C07218=1044.271,328.276,-116.998,172.493,41.338,157.946
C07219=1044.264,328.029,-116.963,172.488,41.335,157.945
C07220=1044.256,327.782,-116.928,172.484,41.332,157.944
C07221=1044.249,327.534,-116.893,172.479,41.328,157.943
C07222=1044.242,327.286,-116.857,172.474,41.325,157.942
C07223=1044.235,327.039,-116.823,172.470,41.322,157.941
C07224=1044.227,326.791,-116.787,172.466,41.319,157.940
C07225=1044.220,326.544,-116.753,172.461,41.316,157.939
C07226=1044.213,326.297,-116.718,172.457,41.313,157.938
C07227=1044.206,326.049,-116.683,172.453,41.310,157.937
C07228=1044.198,325.802,-116.648,172.449,41.307,157.936
C07229=1044.191,325.554,-116.613,172.444,41.304,157.935
C07230=1044.184,325.307,-116.578,172.440,41.301,157.934
C07231=1044.177,325.060,-116.543,172.436,41.298,157.933
C07232=1044.170,324.812,-116.509,172.431,41.295,157.932
C07233=1044.163,324.564,-116.474,172.427,41.292,157.931
C07234=1044.156,324.317,-116.438,172.423,41.289,157.930
C07235=1044.148,324.070,-116.404,172.419,41.286,157.929
C07236=1044.141,323.822,-116.369,172.414,41.283,157.929
C07237=1044.134,323.575,-116.335,172.410,41.280,157.928
C07238=1044.128,323.327,-116.300,172.406,41.277,157.927
C07239=1044.120,323.080,-116.265,172.401,41.274,157.926
C07240=1044.113,322.833,-116.230,172.398,41.271,157.925
C07241=1044.106,322.584,-116.195,172.392,41.268,157.924
C07242=1044.099,322.337,-116.161,172.388,41.265,157.923
C07243=1044.092,322.090,-116.126,172.384,41.262,157.922
C07244=1044.085,321.842,-116.092,172.380,41.259,157.921
C07245=1044.078,321.595,-116.057,172.376,41.256,157.920
C07246=1044.071,321.347,-116.023,172.371,41.254,157.920
C07247=1044.064,321.100,-115.988,172.367,41.250,157.919
C07248=1044.056,320.853,-115.953,172.363,41.247,157.918
C07249=1044.050,320.605,-115.919,172.359,41.245,157.917
C07250=1044.042,320.358,-115.884,172.355,41.241,157.916
C07251=1044.036,320.110,-115.850,172.350,41.238,157.915
C07252=1044.027,319.780,-115.803,172.345,41.235,157.914
C07253=1044.017,319.450,-115.758,172.340,41.231,157.913
C07254=1044.008,319.121,-115.712,172.334,41.227,157.911
C07255=1043.999,318.792,-115.666,172.329,41.223,157.910
C07256=1043.993,318.544,-115.632,172.325,41.220,157.909
C07257=1043.985,318.297,-115.597,172.320,41.217,157.909
C07258=1043.979,318.049,-115.563,172.316,41.214,157.908
C07259=1043.972,317.801,-115.529,172.312,41.211,157.907
C07260=1043.965,317.554,-115.494,172.308,41.208,157.906
C07261=1043.958,317.306,-115.460,172.304,41.205,157.905
C07262=1043.951,317.058,-115.426,172.300,41.203,157.904
C07263=1043.944,316.811,-115.391,172.296,41.200,157.903
C07264=1043.938,316.564,-115.357,172.292,41.197,157.902
C07265=1043.931,316.316,-115.323,172.288,41.194,157.901
C07266=1043.924,316.068,-115.289,172.284,41.191,157.901
C07267=1043.917,315.821,-115.254,172.280,41.188,157.900
C07268=1043.910,315.573,-115.220,172.275,41.185,157.899
C07269=1043.904,315.326,-115.186,172.271,41.182,157.898
C07270=1043.897,315.078,-115.152,172.267,41.180,157.897
C07271=1043.890,314.831,-115.117,172.263,41.177,157.896
C07272=1043.882,314.584,-115.084,172.259,41.174,157.895
C07273=1043.877,314.336,-115.050,172.255,41.171,157.895
C07274=1043.869,314.089,-115.016,172.251,41.168,157.894
C07275=1043.863,313.841,-114.981,172.247,41.165,157.893
C07276=1043.856,313.593,-114.947,172.243,41.162,157.892
C07277=1043.850,313.346,-114.913,172.239,41.160,157.891
C07278=1043.843,313.098,-114.880,172.236,41.157,157.890
C07279=1043.836,312.850,-114.845,172.231,41.154,157.889
C07280=1043.830,312.603,-114.812,172.228,41.151,157.889
C07281=1043.822,312.355,-114.778,172.224,41.149,157.888
C07282=1043.815,312.108,-114.744,172.220,41.145,157.887
C07283=1043.808,311.860,-114.710,172.216,41.143,157.886
C07284=1043.801,311.612,-114.676,172.212,41.140,157.885
C07285=1043.794,311.365,-114.643,172.208,41.138,157.884
C07286=1043.787,311.118,-114.609,172.204,41.135,157.884
C07287=1043.780,310.870,-114.576,172.200,41.132,157.883
C07288=1043.773,310.622,-114.542,172.196,41.130,157.882
C07289=1043.766,310.375,-114.509,172.192,41.127,157.881
C07290=1043.759,310.127,-114.475,172.189,41.125,157.880
C07291=1043.751,309.879,-114.442,172.185,41.122,157.880
C07292=1043.745,309.632,-114.409,172.181,41.119,157.879
C07293=1043.738,309.385,-114.375,172.177,41.116,157.878
C07294=1043.731,309.136,-114.342,172.173,41.113,157.877
C07295=1043.724,308.889,-114.309,172.169,41.111,157.876
C07296=1043.717,308.642,-114.275,172.165,41.108,157.875
C07297=1043.710,308.393,-114.242,172.161,41.106,157.875
C07298=1043.703,308.146,-114.208,172.157,41.103,157.874
C07299=1043.696,307.898,-114.176,172.153,41.100,157.873
C07300=1043.689,307.651,-114.142,172.149,41.098,157.872
C07301=1043.682,307.404,-114.108,172.146,41.095,157.872
C07302=1043.675,307.155,-114.075,172.142,41.093,157.871
C07303=1043.669,306.908,-114.042,172.138,41.090,157.870
C07304=1043.662,306.660,-114.009,172.134,41.087,157.869
C07305=1043.654,306.412,-113.975,172.130,41.085,157.868
C07306=1043.647,306.165,-113.943,172.126,41.082,157.868
C07307=1043.640,305.918,-113.909,172.122,41.079,157.867
C07308=1043.632,305.593,-113.865,172.117,41.076,157.866
C07309=1043.623,305.268,-113.822,172.112,41.073,157.865
C07310=1043.614,304.942,-113.778,172.107,41.070,157.864
C07311=1043.605,304.618,-113.735,172.102,41.066,157.863
C07312=1043.597,304.370,-113.702,172.099,41.063,157.862
C07313=1043.591,304.123,-113.669,172.095,41.060,157.861
C07314=1043.584,303.875,-113.636,172.091,41.058,157.860
C07315=1043.578,303.627,-113.603,172.087,41.056,157.860
C07316=1043.570,303.379,-113.569,172.084,41.053,157.859
C07317=1043.564,303.132,-113.536,172.080,41.051,157.858
C07318=1043.557,302.885,-113.504,172.076,41.048,157.857
C07319=1043.550,302.636,-113.471,172.072,41.045,157.856
C07320=1043.544,302.389,-113.437,172.068,41.043,157.856
C07321=1043.537,302.141,-113.404,172.065,41.040,157.855
C07322=1043.530,301.893,-113.372,172.061,41.037,157.854
C07323=1043.523,301.645,-113.339,172.057,41.035,157.853
C07324=1043.516,301.398,-113.306,172.054,41.032,157.853
C07325=1043.510,301.151,-113.273,172.050,41.030,157.852
C07326=1043.503,300.903,-113.240,172.046,41.027,157.851
C07327=1043.497,300.655,-113.207,172.042,41.025,157.850
C07328=1043.490,300.407,-113.174,172.039,41.022,157.850
C07329=1043.483,300.159,-113.142,172.035,41.019,157.849
C07330=1043.476,299.912,-113.108,172.031,41.017,157.848
C07331=1043.469,299.664,-113.075,172.028,41.015,157.847
C07332=1043.463,299.416,-113.043,172.024,41.012,157.847
C07333=1043.457,299.169,-113.010,172.020,41.009,157.846
C07334=1043.449,298.921,-112.977,172.017,41.007,157.845
C07335=1043.443,298.673,-112.945,172.013,41.004,157.844
C07336=1043.436,298.426,-112.912,172.009,41.001,157.843
C07337=1043.430,298.178,-112.879,172.006,40.999,157.843
C07338=1043.423,297.930,-112.847,172.002,40.997,157.842
C07339=1043.416,297.683,-112.814,171.999,40.994,157.841
C07340=1043.410,297.435,-112.781,171.995,40.991,157.840
C07341=1043.403,297.187,-112.748,171.991,40.989,157.840
C07342=1043.397,296.939,-112.715,171.988,40.987,157.839
C07343=1043.390,296.692,-112.683,171.985,40.984,157.838
C07344=1043.383,296.444,-112.650,171.981,40.981,157.837
C07345=1043.377,296.197,-112.618,171.977,40.979,157.837
C07346=1043.371,295.948,-112.585,171.973,40.976,157.836
C07347=1043.364,295.700,-112.553,171.970,40.974,157.835
C07348=1043.357,295.453,-112.520,171.967,40.971,157.834
C07349=1043.350,295.206,-112.488,171.963,40.969,157.834
C07350=1043.343,294.957,-112.455,171.959,40.966,157.833
C07351=1043.337,294.709,-112.424,171.956,40.964,157.832
C07352=1043.330,294.462,-112.391,171.952,40.962,157.832
C07353=1043.323,294.214,-112.359,171.949,40.959,157.831
C07354=1043.317,293.966,-112.326,171.945,40.957,157.830
C07355=1043.310,293.718,-112.294,171.941,40.954,157.829
C07356=1043.303,293.471,-112.261,171.938,40.951,157.829
C07357=1043.297,293.223,-112.230,171.934,40.949,157.828
C07358=1043.289,292.975,-112.197,171.931,40.947,157.827
C07359=1043.283,292.727,-112.165,171.927,40.945,157.827
C07360=1043.276,292.479,-112.133,171.924,40.942,157.826
C07361=1043.269,292.232,-112.101,171.920,40.940,157.825
C07362=1043.263,291.984,-112.069,171.916,40.937,157.824
C07363=1043.255,291.736,-112.037,171.914,40.935,157.824
C07364=1043.247,291.427,-111.997,171.909,40.932,157.823
C07365=1043.239,291.119,-111.957,171.905,40.929,157.822
C07366=1043.231,290.810,-111.917,171.900,40.926,157.821
C07367=1043.223,290.502,-111.877,171.896,40.923,157.820
C07368=1043.215,290.254,-111.846,171.892,40.921,157.820
C07369=1043.208,290.006,-111.813,171.889,40.918,157.819
C07370=1043.202,289.758,-111.781,171.886,40.916,157.818
C07371=1043.196,289.510,-111.750,171.882,40.914,157.817
C07372=1043.188,289.263,-111.718,171.879,40.911,157.817
C07373=1043.182,289.015,-111.686,171.875,40.909,157.816
C07374=1043.176,288.767,-111.654,171.871,40.906,157.815
C07375=1043.169,288.520,-111.622,171.869,40.904,157.815
C07376=1043.162,288.272,-111.591,171.865,40.902,157.814
C07377=1043.155,288.023,-111.559,171.861,40.900,157.813
C07378=1043.148,287.775,-111.526,171.859,40.897,157.813
C07379=1043.142,287.528,-111.495,171.855,40.895,157.812
C07380=1043.135,287.280,-111.463,171.851,40.893,157.811
C07381=1043.128,287.032,-111.432,171.848,40.890,157.810
C07382=1043.121,286.785,-111.400,171.844,40.888,157.810
C07383=1043.114,286.537,-111.368,171.841,40.886,157.809
C07384=1043.108,286.289,-111.337,171.838,40.883,157.808
C07385=1043.101,286.041,-111.305,171.834,40.881,157.808
C07386=1043.094,285.793,-111.274,171.831,40.879,157.807
C07387=1043.088,285.545,-111.243,171.828,40.877,157.807
C07388=1043.081,285.297,-111.211,171.824,40.874,157.806
C07389=1043.074,285.049,-111.180,171.820,40.872,157.805
C07390=1043.067,284.802,-111.148,171.818,40.870,157.804
C07391=1043.061,284.554,-111.116,171.814,40.867,157.804
C07392=1043.054,284.306,-111.084,171.811,40.865,157.803
C07393=1043.048,284.058,-111.053,171.807,40.863,157.802
C07394=1043.041,283.810,-111.021,171.804,40.861,157.802
C07395=1043.034,283.562,-110.990,171.801,40.858,157.801
C07396=1043.027,283.314,-110.958,171.797,40.856,157.800
C07397=1043.021,283.066,-110.927,171.794,40.854,157.800
C07398=1043.014,282.818,-110.895,171.791,40.851,157.799
C07399=1043.007,282.570,-110.864,171.787,40.849,157.798
C07400=1043.001,282.322,-110.833,171.784,40.847,157.798
C07401=1042.994,282.074,-110.802,171.781,40.845,157.797
C07402=1042.987,281.826,-110.770,171.778,40.842,157.796
C07403=1042.981,281.578,-110.739,171.774,40.840,157.796
C07404=1042.974,281.330,-110.708,171.770,40.838,157.795
C07405=1042.967,281.082,-110.676,171.768,40.836,157.794
C07406=1042.961,280.835,-110.645,171.764,40.833,157.794
C07407=1042.954,280.587,-110.613,171.761,40.831,157.793
C07408=1042.947,280.338,-110.583,171.758,40.829,157.792
C07409=1042.941,280.090,-110.551,171.755,40.827,157.792
C07410=1042.935,279.843,-110.520,171.751,40.824,157.791
C07411=1042.928,279.595,-110.489,171.748,40.822,157.790
C07412=1042.921,279.347,-110.457,171.745,40.820,157.790
C07413=1042.915,279.099,-110.427,171.742,40.817,157.789
C07414=1042.908,278.851,-110.395,171.738,40.815,157.789
C07415=1042.900,278.603,-110.364,171.734,40.813,157.788
C07416=1042.894,278.355,-110.334,171.732,40.811,157.787
C07417=1042.887,278.107,-110.302,171.728,40.808,157.787
C07418=1042.881,277.860,-110.271,171.725,40.806,157.786
C07419=1042.874,277.611,-110.241,171.722,40.804,157.785
C07420=1042.866,277.314,-110.203,171.718,40.802,157.785
C07421=1042.858,277.017,-110.166,171.714,40.799,157.784
C07422=1042.850,276.721,-110.129,171.710,40.796,157.783
C07423=1042.842,276.424,-110.092,171.706,40.793,157.782
C07424=1042.835,276.177,-110.062,171.704,40.791,157.782
C07425=1042.829,275.928,-110.031,171.700,40.789,157.781
C07426=1042.822,275.680,-109.999,171.697,40.787,157.780
C07427=1042.815,275.432,-109.968,171.694,40.785,157.780
C07428=1042.808,275.184,-109.938,171.691,40.783,157.779
C07429=1042.803,274.936,-109.908,171.687,40.781,157.778
C07430=1042.796,274.688,-109.876,171.685,40.778,157.778
C07431=1042.789,274.440,-109.845,171.681,40.776,157.777
C07432=1042.782,274.192,-109.815,171.678,40.774,157.777
C07433=1042.775,273.944,-109.784,171.674,40.772,157.776
C07434=1042.769,273.697,-109.753,171.672,40.769,157.775
C07435=1042.762,273.448,-109.723,171.668,40.767,157.775
C07436=1042.756,273.200,-109.692,171.665,40.765,157.774
C07437=1042.749,272.952,-109.661,171.662,40.763,157.773
C07438=1042.743,272.705,-109.631,171.659,40.761,157.773
C07439=1042.736,272.456,-109.600,171.656,40.759,157.772
C07440=1042.729,272.208,-109.569,171.653,40.756,157.771
C07441=1042.722,271.960,-109.538,171.650,40.754,157.771
C07442=1042.716,271.712,-109.508,171.646,40.752,157.770
C07443=1042.709,271.464,-109.477,171.644,40.750,157.770
C07444=1042.703,271.216,-109.447,171.640,40.748,157.769
C07445=1042.696,270.968,-109.417,171.637,40.746,157.768
C07446=1042.690,270.720,-109.386,171.635,40.744,157.768
C07447=1042.682,270.472,-109.355,171.631,40.741,157.767
C07448=1042.676,270.224,-109.325,171.628,40.739,157.767
C07449=1042.669,269.976,-109.295,171.625,40.737,157.766
C07450=1042.663,269.728,-109.264,171.622,40.735,157.765
C07451=1042.656,269.480,-109.234,171.618,40.733,157.765
C07452=1042.650,269.232,-109.204,171.616,40.731,157.764
C07453=1042.642,268.984,-109.173,171.613,40.728,157.763
C07454=1042.636,268.736,-109.142,171.609,40.726,157.763
C07455=1042.629,268.488,-109.112,171.607,40.724,157.762
C07456=1042.623,268.240,-109.082,171.603,40.723,157.762
C07457=1042.616,267.991,-109.051,171.600,40.720,157.761
C07458=1042.610,267.744,-109.021,171.598,40.718,157.761
C07459=1042.603,267.495,-108.991,171.594,40.716,157.760
C07460=1042.596,267.247,-108.960,171.591,40.714,157.759
C07461=1042.590,266.999,-108.931,171.588,40.712,157.759
C07462=1042.583,266.751,-108.900,171.585,40.710,157.758
C07463=1042.576,266.503,-108.870,171.582,40.707,157.757
C07464=1042.565,266.110,-108.822,171.577,40.704,157.756
C07465=1042.555,265.716,-108.775,171.572,40.701,157.756
C07466=1042.544,265.323,-108.727,171.567,40.698,157.755
C07467=1042.534,264.929,-108.679,171.563,40.695,157.754
C07468=1042.527,264.681,-108.649,171.560,40.692,157.753
C07469=1042.521,264.433,-108.619,171.557,40.690,157.752
C07470=1042.514,264.185,-108.589,171.554,40.688,157.752
C07471=1042.507,263.937,-108.559,171.551,40.686,157.751
C07472=1042.497,263.542,-108.511,171.546,40.683,157.750
C07473=1042.486,263.147,-108.463,171.542,40.679,157.749
C07474=1042.476,262.752,-108.416,171.537,40.676,157.748
C07475=1042.466,262.357,-108.367,171.532,40.672,157.747
C07476=1042.459,262.109,-108.338,171.529,40.671,157.747
C07477=1042.452,261.861,-108.308,171.526,40.669,157.746
C07478=1042.445,261.612,-108.278,171.523,40.667,157.746
C07479=1042.439,261.364,-108.249,171.520,40.664,157.745
C07480=1042.432,261.116,-108.219,171.518,40.663,157.745
C07481=1042.425,260.869,-108.189,171.514,40.661,157.744
C07482=1042.418,260.620,-108.160,171.511,40.658,157.743
C07483=1042.411,260.371,-108.130,171.509,40.657,157.743
C07484=1042.405,260.123,-108.101,171.505,40.655,157.742
C07485=1042.398,259.875,-108.071,171.502,40.652,157.742
C07486=1042.391,259.627,-108.041,171.500,40.651,157.741
C07487=1042.384,259.379,-108.011,171.496,40.649,157.741
C07488=1042.377,259.131,-107.983,171.494,40.647,157.740
C07489=1042.370,258.883,-107.953,171.491,40.644,157.739
C07490=1042.364,258.635,-107.924,171.489,40.643,157.739
C07491=1042.357,258.386,-107.894,171.485,40.641,157.738
C07492=1042.351,258.138,-107.865,171.482,40.638,157.738
C07493=1042.343,257.890,-107.834,171.480,40.637,157.737
C07494=1042.337,257.642,-107.805,171.476,40.635,157.737
C07495=1042.330,257.394,-107.775,171.473,40.632,157.736
C07496=1042.324,257.146,-107.746,171.471,40.631,157.736
C07497=1042.317,256.897,-107.717,171.468,40.629,157.735
C07498=1042.310,256.649,-107.687,171.465,40.627,157.734
C07499=1042.303,256.400,-107.658,171.462,40.625,157.734
C07500=1042.297,256.153,-107.628,171.459,40.623,157.733
C07501=1042.291,255.905,-107.599,171.456,40.621,157.733
C07502=1042.283,255.656,-107.570,171.453,40.618,157.732
C07503=1042.276,255.409,-107.540,171.451,40.617,157.732
C07504=1042.270,255.160,-107.511,171.448,40.615,157.731
C07505=1042.263,254.912,-107.482,171.445,40.612,157.730
C07506=1042.257,254.664,-107.452,171.442,40.611,157.730
C07507=1042.250,254.415,-107.423,171.439,40.609,157.729
C07508=1042.244,254.167,-107.394,171.436,40.606,157.729
C07509=1042.237,253.918,-107.364,171.434,40.605,157.728
C07510=1042.230,253.671,-107.335,171.430,40.603,157.728
C07511=1042.224,253.423,-107.305,171.428,40.600,157.727
C07512=1042.217,253.174,-107.276,171.425,40.599,157.726
C07513=1042.210,252.926,-107.248,171.423,40.597,157.726
C07514=1042.204,252.679,-107.218,171.420,40.594,157.725
C07515=1042.197,252.430,-107.188,171.416,40.592,157.725
C07516=1042.191,252.182,-107.159,171.414,40.591,157.724
C07517=1042.184,251.934,-107.130,171.411,40.588,157.724
C07518=1042.177,251.685,-107.101,171.408,40.586,157.723
C07519=1042.171,251.437,-107.071,171.406,40.585,157.723
C07520=1042.165,251.189,-107.042,171.402,40.583,157.722
C07521=1042.158,250.940,-107.013,171.400,40.580,157.721
C07522=1042.151,250.692,-106.984,171.397,40.579,157.721
C07523=1042.145,250.444,-106.955,171.394,40.576,157.720
C07524=1042.138,250.196,-106.926,171.392,40.574,157.720
C07525=1042.131,249.947,-106.897,171.389,40.572,157.719
C07526=1042.125,249.699,-106.868,171.386,40.571,157.719
C07527=1042.119,249.451,-106.839,171.383,40.568,157.718
C07528=1042.110,249.157,-106.804,171.380,40.566,157.717
C07529=1042.103,248.864,-106.769,171.377,40.563,157.717
C07530=1042.095,248.571,-106.735,171.374,40.561,157.716
C07531=1042.088,248.276,-106.701,171.370,40.558,157.715
C07532=1042.082,248.028,-106.672,171.368,40.557,157.715
C07533=1042.075,247.780,-106.643,171.365,40.555,157.714
C07534=1042.068,247.532,-106.614,171.362,40.552,157.714
C07535=1042.062,247.284,-106.585,171.360,40.551,157.713
C07536=1042.056,247.035,-106.556,171.357,40.548,157.713
C07537=1042.049,246.787,-106.527,171.354,40.546,157.712
C07538=1042.042,246.538,-106.498,171.351,40.545,157.711
C07539=1042.036,246.290,-106.469,171.348,40.542,157.711
C07540=1042.029,246.043,-106.440,171.346,40.540,157.710
C07541=1042.023,245.794,-106.411,171.343,40.538,157.710
C07542=1042.017,245.546,-106.382,171.341,40.536,157.709
C07543=1042.010,245.298,-106.353,171.338,40.534,157.709
C07544=1042.004,245.049,-106.324,171.335,40.532,157.708
C07545=1041.997,244.801,-106.296,171.333,40.530,157.708
C07546=1041.991,244.553,-106.267,171.330,40.528,157.707
C07547=1041.984,244.305,-106.238,171.328,40.526,157.706
C07548=1041.977,244.057,-106.209,171.325,40.524,157.706
C07549=1041.971,243.807,-106.181,171.321,40.522,157.705
C07550=1041.964,243.559,-106.152,171.319,40.520,157.705
C07551=1041.958,243.311,-106.123,171.316,40.518,157.704
C07552=1041.951,243.064,-106.095,171.314,40.516,157.704
C07553=1041.945,242.815,-106.066,171.311,40.514,157.703
C07554=1041.938,242.567,-106.037,171.308,40.512,157.703
C07555=1041.932,242.319,-106.009,171.306,40.511,157.702
C07556=1041.925,242.069,-105.980,171.303,40.508,157.701
C07557=1041.918,241.822,-105.952,171.301,40.506,157.701
C07558=1041.912,241.573,-105.923,171.298,40.504,157.700
C07559=1041.906,241.325,-105.894,171.296,40.502,157.700
C07560=1041.899,241.077,-105.866,171.293,40.501,157.699
C07561=1041.892,240.829,-105.838,171.290,40.498,157.699
C07562=1041.886,240.580,-105.809,171.288,40.497,157.698
C07563=1041.878,240.332,-105.780,171.285,40.494,157.698
C07564=1041.872,240.083,-105.752,171.282,40.492,157.697
C07565=1041.865,239.835,-105.724,171.279,40.491,157.697
C07566=1041.859,239.587,-105.696,171.276,40.488,157.696
C07567=1041.852,239.339,-105.667,171.274,40.487,157.696
C07568=1041.846,239.090,-105.639,171.271,40.485,157.695
C07569=1041.839,238.842,-105.611,171.269,40.483,157.695
C07570=1041.833,238.594,-105.582,171.266,40.481,157.694
C07571=1041.826,238.346,-105.554,171.264,40.479,157.693
C07572=1041.819,238.097,-105.526,171.261,40.477,157.693
C07573=1041.812,237.849,-105.497,171.259,40.475,157.692
C07574=1041.806,237.600,-105.469,171.256,40.473,157.692
C07575=1041.799,237.352,-105.441,171.253,40.471,157.691
C07576=1041.792,237.104,-105.413,171.251,40.469,157.691
C07577=1041.786,236.855,-105.385,171.248,40.467,157.690
C07578=1041.779,236.607,-105.357,171.246,40.465,157.690
C07579=1041.772,236.359,-105.328,171.243,40.464,157.689
C07580=1041.766,236.110,-105.300,171.241,40.461,157.689
C07581=1041.759,235.862,-105.272,171.238,40.460,157.688
C07582=1041.753,235.614,-105.244,171.235,40.458,157.688
C07583=1041.746,235.365,-105.216,171.233,40.456,157.687
C07584=1041.738,235.065,-105.182,171.230,40.453,157.686
C07585=1041.730,234.766,-105.148,171.227,40.451,157.686
C07586=1041.722,234.467,-105.114,171.224,40.449,157.685
C07587=1041.714,234.167,-105.080,171.220,40.447,157.685
C07588=1041.707,233.919,-105.052,171.218,40.444,157.684
C07589=1041.701,233.671,-105.024,171.216,40.443,157.684
C07590=1041.695,233.422,-104.996,171.214,40.440,157.683
C07591=1041.689,233.174,-104.968,171.211,40.439,157.682
C07592=1041.682,232.926,-104.940,171.208,40.436,157.682
C07593=1041.675,232.678,-104.912,171.206,40.434,157.681
C07594=1041.669,232.429,-104.884,171.203,40.433,157.681
C07595=1041.662,232.181,-104.856,171.201,40.430,157.680
C07596=1041.656,231.932,-104.828,171.198,40.429,157.680
C07597=1041.649,231.684,-104.800,171.196,40.426,157.679
C07598=1041.642,231.436,-104.772,171.193,40.425,157.679
C07599=1041.635,231.187,-104.744,171.190,40.422,157.678
C07600=1041.629,230.939,-104.717,171.188,40.421,157.678
C07601=1041.623,230.690,-104.688,171.185,40.419,157.677
C07602=1041.616,230.442,-104.660,171.183,40.417,157.677
C07603=1041.609,230.193,-104.633,171.180,40.415,157.676
C07604=1041.603,229.945,-104.605,171.178,40.413,157.676
C07605=1041.596,229.696,-104.577,171.175,40.411,157.675
C07606=1041.589,229.448,-104.550,171.174,40.409,157.675
C07607=1041.583,229.200,-104.522,171.171,40.407,157.674
C07608=1041.577,228.952,-104.494,171.168,40.405,157.674
C07609=1041.570,228.703,-104.467,171.166,40.403,157.673
C07610=1041.563,228.455,-104.439,171.163,40.401,157.672
C07611=1041.557,228.206,-104.411,171.161,40.400,157.672
C07612=1041.550,227.958,-104.384,171.158,40.397,157.671
C07613=1041.543,227.710,-104.356,171.156,40.396,157.671
C07614=1041.536,227.461,-104.328,171.153,40.394,157.670
C07615=1041.530,227.213,-104.300,171.151,40.392,157.670
C07616=1041.523,226.964,-104.273,171.148,40.390,157.669
C07617=1041.516,226.716,-104.245,171.147,40.388,157.669
C07618=1041.509,226.467,-104.218,171.144,40.386,157.668
C07619=1041.503,226.219,-104.191,171.141,40.384,157.668
C07620=1041.497,225.971,-104.163,171.139,40.382,157.667
C07621=1041.490,225.722,-104.136,171.136,40.380,157.667
C07622=1041.483,225.474,-104.108,171.134,40.378,157.666
C07623=1041.476,225.226,-104.080,171.131,40.376,157.666
C07624=1041.470,224.977,-104.052,171.129,40.375,157.665
C07625=1041.463,224.728,-104.025,171.126,40.373,157.665
C07626=1041.456,224.480,-103.998,171.125,40.371,157.664
C07627=1041.450,224.232,-103.971,171.122,40.369,157.664
C07628=1041.443,223.984,-103.943,171.120,40.367,157.663
C07629=1041.437,223.735,-103.916,171.117,40.365,157.663
C07630=1041.430,223.486,-103.888,171.114,40.363,157.662
C07631=1041.424,223.238,-103.861,171.112,40.361,157.662
C07632=1041.417,222.990,-103.833,171.109,40.359,157.661
C07633=1041.410,222.741,-103.807,171.108,40.357,157.661
C07634=1041.404,222.493,-103.779,171.105,40.355,157.660
C07635=1041.397,222.244,-103.752,171.103,40.353,157.660
C07636=1041.390,221.996,-103.724,171.100,40.352,157.659
C07637=1041.385,221.748,-103.697,171.098,40.349,157.659
C07638=1041.378,221.499,-103.669,171.095,40.348,157.658
C07639=1041.370,221.251,-103.642,171.094,40.345,157.658
C07640=1041.362,220.944,-103.608,171.090,40.343,157.657
C07641=1041.354,220.637,-103.575,171.087,40.340,157.656
C07642=1041.346,220.330,-103.541,171.084,40.338,157.656
C07643=1041.338,220.023,-103.507,171.082,40.336,157.655
C07644=1041.332,219.775,-103.481,171.079,40.334,157.655
C07645=1041.325,219.526,-103.453,171.077,40.332,157.654
C07646=1041.318,219.278,-103.426,171.074,40.330,157.654
C07647=1041.312,219.029,-103.399,171.072,40.328,157.653
C07648=1041.305,218.780,-103.372,171.070,40.326,157.653
C07649=1041.298,218.533,-103.345,171.068,40.325,157.652
C07650=1041.292,218.284,-103.318,171.065,40.322,157.651
C07651=1041.285,218.035,-103.291,171.063,40.321,157.651
C07652=1041.278,217.786,-103.264,171.060,40.318,157.650
C07653=1041.271,217.539,-103.237,171.059,40.317,157.650
C07654=1041.265,217.290,-103.210,171.056,40.315,157.650
C07655=1041.258,217.041,-103.184,171.053,40.313,157.649
C07656=1041.251,216.793,-103.156,171.051,40.311,157.649
C07657=1041.246,216.544,-103.129,171.048,40.309,157.648
C07658=1041.238,216.296,-103.102,171.047,40.307,157.648
C07659=1041.232,216.047,-103.075,171.044,40.305,157.647
C07660=1041.225,215.800,-103.048,171.042,40.303,157.646
C07661=1041.219,215.551,-103.021,171.039,40.302,157.646
C07662=1041.211,215.302,-102.995,171.038,40.299,157.645
C07663=1041.205,215.054,-102.968,171.035,40.298,157.645
C07664=1041.199,214.805,-102.941,171.033,40.295,157.644
C07665=1041.192,214.556,-102.914,171.030,40.294,157.644
C07666=1041.186,214.309,-102.887,171.029,40.292,157.644
C07667=1041.179,214.060,-102.860,171.026,40.290,157.643
C07668=1041.172,213.811,-102.833,171.024,40.288,157.642
C07669=1041.165,213.563,-102.807,171.021,40.286,157.642
C07670=1041.159,213.314,-102.780,171.019,40.284,157.641
C07671=1041.152,213.065,-102.753,171.017,40.282,157.641
C07672=1041.146,212.818,-102.726,171.014,40.280,157.640
C07673=1041.139,212.569,-102.699,171.013,40.278,157.640
C07674=1041.132,212.320,-102.672,171.010,40.276,157.639
C07675=1041.127,212.072,-102.646,171.008,40.274,157.639
C07676=1041.119,211.823,-102.618,171.005,40.272,157.638
C07677=1041.113,211.575,-102.592,171.004,40.270,157.638
C07678=1041.106,211.326,-102.565,171.001,40.268,157.637
C07679=1041.099,211.078,-102.539,170.999,40.266,157.637
C07680=1041.093,210.829,-102.512,170.997,40.264,157.636
C07681=1041.086,210.581,-102.485,170.995,40.262,157.636
C07682=1041.080,210.333,-102.459,170.992,40.261,157.635
C07683=1041.073,210.084,-102.432,170.989,40.258,157.635
C07684=1041.066,209.835,-102.406,170.988,40.257,157.634
C07685=1041.060,209.587,-102.379,170.985,40.254,157.634
C07686=1041.053,209.338,-102.353,170.983,40.253,157.633
C07687=1041.047,209.090,-102.327,170.981,40.250,157.633
C07688=1041.040,208.841,-102.300,170.979,40.249,157.632
C07689=1041.033,208.593,-102.272,170.976,40.247,157.632
C07690=1041.026,208.345,-102.246,170.975,40.245,157.631
C07691=1041.020,208.096,-102.219,170.972,40.243,157.631
C07692=1041.013,207.848,-102.193,170.970,40.241,157.630
C07693=1041.006,207.599,-102.167,170.968,40.239,157.630
C07694=1041.000,207.351,-102.141,170.966,40.237,157.629
C07695=1040.993,207.102,-102.114,170.963,40.235,157.629
C07696=1040.985,206.800,-102.082,170.961,40.233,157.628
C07697=1040.977,206.499,-102.051,170.958,40.231,157.628
C07698=1040.969,206.198,-102.019,170.955,40.228,157.627
C07699=1040.960,205.896,-101.986,170.953,40.226,157.627
C07700=1040.935,204.845,-101.880,170.669,40.123,157.593
C07701=1040.929,204.596,-101.855,170.667,40.121,157.593
C07702=1040.922,204.348,-101.830,170.663,40.120,157.593
C07703=1040.916,204.099,-101.804,170.661,40.119,157.592
C07704=1040.910,203.850,-101.779,170.657,40.118,157.592
C07705=1040.904,203.602,-101.754,170.654,40.117,157.592
C07706=1040.898,203.353,-101.729,170.652,40.116,157.591
C07707=1040.892,203.104,-101.704,170.648,40.114,157.591
C07708=1040.886,202.856,-101.679,170.645,40.113,157.590
C07709=1040.879,202.608,-101.654,170.643,40.112,157.590
C07710=1040.873,202.359,-101.629,170.639,40.111,157.590
C07711=1040.867,202.110,-101.604,170.637,40.110,157.589
C07712=1040.861,201.861,-101.579,170.634,40.109,157.589
C07713=1040.855,201.612,-101.553,170.630,40.108,157.589
C07714=1040.849,201.364,-101.528,170.628,40.106,157.588
C07715=1040.843,201.115,-101.504,170.625,40.105,157.588
C07716=1040.837,200.866,-101.478,170.621,40.104,157.588
C07717=1040.830,200.617,-101.454,170.619,40.103,157.587
C07718=1040.824,200.369,-101.429,170.616,40.102,157.587
C07719=1040.817,200.120,-101.404,170.613,40.101,157.587
C07720=1040.811,199.871,-101.380,170.610,40.099,157.586
C07721=1040.806,199.623,-101.355,170.606,40.098,157.586
C07722=1040.799,199.374,-101.331,170.604,40.097,157.586
C07723=1040.793,199.125,-101.305,170.601,40.096,157.585
C07724=1040.786,198.876,-101.281,170.598,40.095,157.585
C07725=1040.780,198.628,-101.256,170.595,40.094,157.585
C07726=1040.773,198.379,-101.232,170.592,40.093,157.584
C07727=1040.768,198.131,-101.207,170.590,40.092,157.584
C07728=1040.762,197.882,-101.182,170.586,40.091,157.584
C07729=1040.755,197.633,-101.158,170.583,40.090,157.583
C07730=1040.749,197.384,-101.133,170.581,40.089,157.583
C07731=1040.742,197.136,-101.109,170.577,40.088,157.583
C07732=1040.737,196.887,-101.084,170.575,40.087,157.582
C07733=1040.730,196.639,-101.059,170.572,40.086,157.582
C07734=1040.724,196.389,-101.035,170.568,40.085,157.582
C07735=1040.718,196.141,-101.010,170.566,40.084,157.581
C07736=1040.712,195.892,-100.986,170.563,40.083,157.581
C07737=1040.706,195.643,-100.961,170.560,40.082,157.581
C07738=1040.699,195.395,-100.936,170.557,40.081,157.580
C07739=1040.693,195.146,-100.912,170.555,40.080,157.580
C07740=1040.686,194.898,-100.887,170.551,40.079,157.580
C07741=1040.681,194.648,-100.863,170.549,40.078,157.579
C07742=1040.674,194.400,-100.839,170.546,40.077,157.579
C07743=1040.668,194.152,-100.814,170.542,40.076,157.579
C07744=1040.662,193.903,-100.790,170.540,40.075,157.578
C07745=1040.656,193.653,-100.765,170.537,40.074,157.578
C07746=1040.650,193.405,-100.740,170.534,40.073,157.578
C07747=1040.644,193.156,-100.716,170.531,40.072,157.577
C07748=1040.638,192.907,-100.691,170.529,40.071,157.577
C07749=1040.632,192.659,-100.668,170.526,40.070,157.577
C07750=1040.625,192.410,-100.642,170.523,40.069,157.577
C07751=1040.619,192.162,-100.619,170.520,40.068,157.576
C07752=1040.613,191.912,-100.594,170.518,40.067,157.576
C07753=1040.607,191.664,-100.570,170.514,40.066,157.576
C07754=1040.601,191.416,-100.545,170.512,40.065,157.575
C07755=1040.595,191.167,-100.521,170.509,40.064,157.575
C07756=1040.589,190.917,-100.497,170.506,40.063,157.575
C07757=1040.583,190.669,-100.473,170.503,40.062,157.574
C07758=1040.577,190.420,-100.448,170.501,40.061,157.574
C07759=1040.570,190.172,-100.424,170.498,40.060,157.574
C07760=1040.564,189.923,-100.399,170.495,40.059,157.573
C07761=1040.557,189.638,-100.372,170.492,40.058,157.573
C07762=1040.551,189.354,-100.344,170.488,40.057,157.573
C07763=1040.544,189.070,-100.317,170.485,40.056,157.572
C07764=1040.537,188.785,-100.288,170.482,40.055,157.572
C07765=1040.531,188.537,-100.264,170.480,40.054,157.572
C07766=1040.525,188.287,-100.240,170.476,40.053,157.571
C07767=1040.519,188.039,-100.216,170.474,40.052,157.571
C07768=1040.513,187.790,-100.192,170.471,40.051,157.571
C07769=1040.507,187.542,-100.168,170.468,40.050,157.570
C07770=1040.500,187.293,-100.144,170.465,40.049,157.570
C07771=1040.495,187.044,-100.120,170.463,40.048,157.570
C07772=1040.488,186.795,-100.096,170.460,40.047,157.569
C07773=1040.483,186.546,-100.071,170.457,40.046,157.569
C07774=1040.477,186.297,-100.047,170.455,40.045,157.569
C07775=1040.471,186.049,-100.023,170.452,40.044,157.569
C07776=1040.465,185.800,-99.999,170.449,40.043,157.568
C07777=1040.459,185.551,-99.975,170.446,40.042,157.568
C07778=1040.453,185.302,-99.951,170.444,40.041,157.568
C07779=1040.447,185.054,-99.926,170.441,40.040,157.567
C07780=1040.441,184.805,-99.902,170.438,40.039,157.567
C07781=1040.435,184.556,-99.878,170.436,40.038,157.567
C07782=1040.429,184.307,-99.854,170.432,40.037,157.566
C07783=1040.424,184.059,-99.830,170.430,40.037,157.566
C07784=1040.417,183.810,-99.806,170.427,40.036,157.566
C07785=1040.412,183.561,-99.782,170.425,40.034,157.565
C07786=1040.406,183.313,-99.758,170.422,40.033,157.565
C07787=1040.398,183.064,-99.735,170.419,40.033,157.565
C07788=1040.392,182.815,-99.712,170.417,40.032,157.565
C07789=1040.386,182.566,-99.688,170.413,40.031,157.564
C07790=1040.379,182.317,-99.664,170.411,40.031,157.564
C07791=1040.373,182.068,-99.641,170.408,40.030,157.564
C07792=1040.367,181.819,-99.617,170.406,40.029,157.564
C07793=1040.361,181.571,-99.594,170.403,40.028,157.563
C07794=1040.354,181.322,-99.570,170.400,40.028,157.563
C07795=1040.348,181.073,-99.546,170.397,40.027,157.563
C07796=1040.342,180.824,-99.523,170.395,40.026,157.563
C07797=1040.336,180.575,-99.499,170.392,40.025,157.562
C07798=1040.330,180.327,-99.475,170.389,40.024,157.562
C07799=1040.323,180.078,-99.453,170.387,40.024,157.562
C07800=1040.317,179.830,-99.429,170.384,40.023,157.562
C07801=1040.311,179.580,-99.406,170.382,40.022,157.561
C07802=1040.304,179.332,-99.382,170.378,40.022,157.561
C07803=1040.298,179.083,-99.358,170.376,40.020,157.561
C07804=1040.292,178.834,-99.335,170.373,40.020,157.561
C07805=1040.285,178.585,-99.311,170.371,40.019,157.560
C07806=1040.280,178.336,-99.288,170.368,40.019,157.560
C07807=1040.274,178.088,-99.264,170.365,40.018,157.560
C07808=1040.267,177.838,-99.241,170.363,40.017,157.560
C07809=1040.261,177.590,-99.218,170.360,40.016,157.559
C07810=1040.254,177.340,-99.195,170.357,40.016,157.559
C07811=1040.248,177.092,-99.171,170.354,40.015,157.559
C07812=1040.243,176.843,-99.148,170.352,40.014,157.559
C07813=1040.236,176.594,-99.124,170.350,40.013,157.558
C07814=1040.230,176.345,-99.101,170.346,40.012,157.558
C07815=1040.224,176.096,-99.077,170.344,40.012,157.558
C07816=1040.218,175.848,-99.054,170.341,40.011,157.557
C07817=1040.211,175.600,-99.031,170.339,40.010,157.557
C07818=1040.205,175.350,-99.008,170.336,40.009,157.557
C07819=1040.199,175.102,-98.984,170.333,40.009,157.557
C07820=1040.193,174.853,-98.961,170.331,40.008,157.556
C07821=1040.187,174.603,-98.938,170.329,40.008,157.556
C07822=1040.181,174.355,-98.914,170.325,40.007,157.556
C07823=1040.175,174.106,-98.891,170.323,40.006,157.556
C07824=1040.168,173.857,-98.867,170.320,40.005,157.555
C07825=1040.161,173.573,-98.841,170.318,40.004,157.555
C07826=1040.155,173.287,-98.815,170.315,40.004,157.555
C07827=1040.147,173.003,-98.788,170.311,40.003,157.555
C07828=1040.141,172.718,-98.762,170.309,40.002,157.554
C07829=1040.135,172.470,-98.738,170.306,40.001,157.554
C07830=1040.127,172.220,-98.715,170.303,40.000,157.554
C07831=1040.122,171.971,-98.692,170.301,40.000,157.554
C07832=1040.116,171.723,-98.669,170.298,39.999,157.553
C07833=1040.110,171.474,-98.646,170.296,39.998,157.553
C07834=1040.104,171.225,-98.623,170.293,39.997,157.553
C07835=1040.098,170.976,-98.600,170.290,39.997,157.553
C07836=1040.091,170.728,-98.577,170.288,39.996,157.552
C07837=1040.085,170.479,-98.554,170.286,39.995,157.552
C07838=1040.079,170.229,-98.530,170.283,39.994,157.552
C07839=1040.073,169.980,-98.507,170.280,39.994,157.552
C07840=1040.067,169.732,-98.484,170.278,39.993,157.551
C07841=1040.062,169.483,-98.461,170.275,39.993,157.551
C07842=1040.055,169.235,-98.438,170.273,39.992,157.551
C07843=1040.049,168.985,-98.415,170.270,39.991,157.551
C07844=1040.043,168.736,-98.392,170.267,39.990,157.550
C07845=1040.037,168.488,-98.368,170.265,39.990,157.550
C07846=1040.031,168.239,-98.346,170.263,39.989,157.550
C07847=1040.026,167.990,-98.323,170.259,39.988,157.550
C07848=1040.018,167.741,-98.300,170.257,39.987,157.549
C07849=1040.013,167.492,-98.277,170.255,39.987,157.549
C07850=1040.007,167.243,-98.254,170.253,39.986,157.549
C07851=1040.001,166.994,-98.231,170.250,39.985,157.549
C07852=1039.995,166.746,-98.207,170.247,39.984,157.548
C07853=1039.989,166.497,-98.185,170.245,39.984,157.548
C07854=1039.983,166.248,-98.162,170.242,39.983,157.548
C07855=1039.977,165.999,-98.139,170.240,39.982,157.548
C07856=1039.971,165.750,-98.116,170.237,39.981,157.547
C07857=1039.965,165.501,-98.093,170.235,39.981,157.547
C07858=1039.960,165.252,-98.070,170.232,39.980,157.547
C07859=1039.953,165.003,-98.048,170.230,39.979,157.547
C07860=1039.947,164.755,-98.025,170.228,39.979,157.547
C07861=1039.942,164.506,-98.002,170.225,39.978,157.546
C07862=1039.936,164.257,-97.979,170.222,39.978,157.546
C07863=1039.929,164.008,-97.956,170.220,39.976,157.546
C07864=1039.924,163.759,-97.933,170.218,39.976,157.546
C07865=1039.918,163.510,-97.910,170.215,39.975,157.545
C07866=1039.912,163.261,-97.887,170.212,39.975,157.545
C07867=1039.906,163.012,-97.864,170.210,39.974,157.545
C07868=1039.899,162.763,-97.842,170.208,39.973,157.545
C07869=1039.894,162.514,-97.819,170.205,39.972,157.544
C07870=1039.888,162.265,-97.796,170.202,39.972,157.544
C07871=1039.882,162.017,-97.773,170.200,39.971,157.544
C07872=1039.876,161.768,-97.750,170.198,39.970,157.544
C07873=1039.870,161.519,-97.728,170.195,39.969,157.543
C07874=1039.864,161.270,-97.705,170.193,39.969,157.543
C07875=1039.859,161.021,-97.682,170.190,39.968,157.543
C07876=1039.853,160.772,-97.660,170.188,39.967,157.543
C07877=1039.847,160.523,-97.637,170.186,39.967,157.542
C07878=1039.841,160.274,-97.614,170.183,39.966,157.542
C07879=1039.835,160.025,-97.591,170.180,39.965,157.542
C07880=1039.829,159.777,-97.569,170.178,39.964,157.542
C07881=1039.823,159.527,-97.547,170.176,39.964,157.541
C07882=1039.817,159.279,-97.524,170.174,39.963,157.541
C07883=1039.810,159.030,-97.502,170.170,39.963,157.541
C07884=1039.805,158.781,-97.479,170.168,39.963,157.541
C07885=1039.798,158.532,-97.458,170.166,39.961,157.541
C07886=1039.792,158.283,-97.435,170.164,39.961,157.540
C07887=1039.786,158.035,-97.412,170.161,39.961,157.540
C07888=1039.780,157.785,-97.390,170.158,39.960,157.540
C07889=1039.773,157.500,-97.365,170.156,39.959,157.540
C07890=1039.765,157.214,-97.339,170.153,39.959,157.540
C07891=1039.759,156.930,-97.314,170.151,39.958,157.539
C07892=1039.752,156.644,-97.288,170.147,39.957,157.539
C07893=1039.746,156.395,-97.265,170.145,39.957,157.539
C07894=1039.739,156.147,-97.243,170.142,39.956,157.539
C07895=1039.734,155.897,-97.221,170.140,39.955,157.538
C07896=1039.727,155.649,-97.198,170.138,39.955,157.538
C07897=1039.721,155.399,-97.177,170.135,39.955,157.538
C07898=1039.715,155.150,-97.154,170.133,39.953,157.538
C07899=1039.709,154.902,-97.131,170.130,39.953,157.538
C07900=1039.703,154.653,-97.110,170.128,39.953,157.537
C07901=1039.697,154.404,-97.087,170.126,39.952,157.537
C07902=1039.691,154.155,-97.065,170.124,39.952,157.537
C07903=1039.684,153.906,-97.043,170.121,39.951,157.537
C07904=1039.678,153.657,-97.021,170.118,39.950,157.537
C07905=1039.673,153.408,-96.998,170.116,39.950,157.536
C07906=1039.666,153.159,-96.977,170.114,39.949,157.536
C07907=1039.660,152.910,-96.954,170.112,39.949,157.536
C07908=1039.654,152.661,-96.933,170.108,39.949,157.536
C07909=1039.648,152.412,-96.910,170.106,39.948,157.536
C07910=1039.642,152.163,-96.888,170.104,39.947,157.535
C07911=1039.636,151.915,-96.866,170.102,39.947,157.535
C07912=1039.630,151.666,-96.844,170.100,39.946,157.535
C07913=1039.624,151.416,-96.823,170.096,39.946,157.535
C07914=1039.618,151.168,-96.800,170.094,39.945,157.535
C07915=1039.612,150.918,-96.778,170.092,39.944,157.534
C07916=1039.605,150.670,-96.756,170.090,39.944,157.534
C07917=1039.599,150.421,-96.734,170.088,39.943,157.534
C07918=1039.593,150.171,-96.713,170.086,39.943,157.534
C07919=1039.587,149.922,-96.690,170.082,39.943,157.534
C07920=1039.581,149.673,-96.668,170.080,39.942,157.533
C07921=1039.575,149.424,-96.646,170.078,39.941,157.533
C07922=1039.569,149.176,-96.624,170.076,39.941,157.533
C07923=1039.563,148.927,-96.603,170.074,39.940,157.533
C07924=1039.557,148.678,-96.581,170.070,39.940,157.533
C07925=1039.550,148.429,-96.559,170.068,39.939,157.532
C07926=1039.545,148.180,-96.537,170.066,39.939,157.532
C07927=1039.539,147.930,-96.515,170.064,39.939,157.532
C07928=1039.532,147.682,-96.493,170.062,39.938,157.532
C07929=1039.526,147.433,-96.471,170.059,39.937,157.532
C07930=1039.520,147.184,-96.450,170.056,39.937,157.531
C07931=1039.514,146.935,-96.428,170.054,39.936,157.531
C07932=1039.508,146.686,-96.406,170.052,39.936,157.531
C07933=1039.502,146.437,-96.384,170.050,39.935,157.531
C07934=1039.495,146.188,-96.362,170.048,39.935,157.531
C07935=1039.489,145.939,-96.341,170.046,39.934,157.531
C07936=1039.483,145.690,-96.319,170.042,39.934,157.530
C07937=1039.477,145.442,-96.297,170.040,39.934,157.530
C07938=1039.471,145.192,-96.275,170.038,39.933,157.530
C07939=1039.465,144.943,-96.254,170.036,39.933,157.530
C07940=1039.459,144.694,-96.232,170.034,39.932,157.530
C07941=1039.452,144.445,-96.211,170.032,39.932,157.529
C07942=1039.446,144.196,-96.190,170.028,39.931,157.529
C07943=1039.440,143.947,-96.168,170.026,39.931,157.529
C07944=1039.434,143.698,-96.147,170.024,39.930,157.529
C07945=1039.428,143.450,-96.124,170.022,39.930,157.529
C07946=1039.421,143.200,-96.103,170.020,39.930,157.529
C07947=1039.415,142.951,-96.081,170.018,39.929,157.528
C07948=1039.410,142.703,-96.060,170.015,39.929,157.528
C07949=1039.403,142.454,-96.038,170.012,39.928,157.528
C07950=1039.397,142.204,-96.016,170.010,39.927,157.528
C07951=1039.391,141.955,-95.995,170.008,39.927,157.528
C07952=1039.385,141.706,-95.973,170.006,39.926,157.527
C07953=1039.378,141.421,-95.949,170.003,39.926,157.527
C07954=1039.371,141.135,-95.924,170.000,39.926,157.527
C07955=1039.364,140.850,-95.899,169.998,39.925,157.527
C07956=1039.357,140.564,-95.875,169.995,39.925,157.527
C07957=1039.351,140.315,-95.854,169.993,39.924,157.527
C07958=1039.345,140.066,-95.832,169.991,39.923,157.526
C07959=1039.339,139.817,-95.811,169.988,39.923,157.526
C07960=1039.333,139.567,-95.789,169.986,39.922,157.526
C07961=1039.327,139.319,-95.768,169.984,39.922,157.526
C07962=1039.321,139.070,-95.746,169.981,39.921,157.526
C07963=1039.314,138.821,-95.725,169.979,39.921,157.525
C07964=1039.308,138.572,-95.704,169.977,39.921,157.525
C07965=1039.302,138.323,-95.682,169.974,39.920,157.525
C07966=1039.296,138.074,-95.661,169.972,39.920,157.525
C07967=1039.289,137.825,-95.640,169.970,39.920,157.525
C07968=1039.284,137.577,-95.618,169.968,39.919,157.525
C07969=1039.278,137.327,-95.597,169.966,39.919,157.524
C07970=1039.272,137.077,-95.576,169.964,39.918,157.524
C07971=1039.265,136.829,-95.555,169.961,39.918,157.524
C07972=1039.259,136.580,-95.533,169.958,39.918,157.524
C07973=1039.253,136.331,-95.512,169.956,39.917,157.524
C07974=1039.246,136.082,-95.491,169.954,39.917,157.524
C07975=1039.241,135.833,-95.470,169.952,39.916,157.523
C07976=1039.235,135.584,-95.449,169.950,39.916,157.523
C07977=1039.228,135.335,-95.427,169.948,39.915,157.523
C07978=1039.222,135.086,-95.406,169.945,39.915,157.523
C07979=1039.216,134.836,-95.385,169.942,39.915,157.523
C07980=1039.209,134.588,-95.364,169.940,39.914,157.522
C07981=1039.203,134.338,-95.343,169.938,39.914,157.522
C07982=1039.198,134.090,-95.321,169.936,39.913,157.522
C07983=1039.191,133.840,-95.301,169.934,39.913,157.522
C07984=1039.185,133.591,-95.279,169.932,39.913,157.522
C07985=1039.179,133.343,-95.258,169.929,39.912,157.522
C07986=1039.172,133.094,-95.237,169.927,39.912,157.522
C07987=1039.167,132.845,-95.217,169.925,39.912,157.521
C07988=1039.161,132.595,-95.195,169.923,39.911,157.521
C07989=1039.154,132.346,-95.174,169.921,39.911,157.521
C07990=1039.149,132.097,-95.153,169.918,39.910,157.521
C07991=1039.143,131.848,-95.132,169.916,39.910,157.521
C07992=1039.136,131.599,-95.111,169.913,39.909,157.521
C07993=1039.131,131.350,-95.090,169.911,39.909,157.520
C07994=1039.124,131.101,-95.068,169.909,39.908,157.520
C07995=1039.118,130.851,-95.048,169.907,39.908,157.520
C07996=1039.112,130.603,-95.027,169.905,39.908,157.520
C07997=1039.106,130.353,-95.007,169.903,39.908,157.520
C07998=1039.099,130.104,-94.985,169.901,39.907,157.520
C07999=1039.092,129.856,-94.965,169.898,39.907,157.519
C08000=1039.087,129.606,-94.944,169.895,39.906,157.519
C08001=1039.080,129.358,-94.923,169.893,39.907,157.519
C08002=1039.074,129.108,-94.902,169.891,39.906,157.519
C08003=1039.068,128.860,-94.881,169.889,39.906,157.519
C08004=1039.062,128.611,-94.861,169.887,39.905,157.519
C08005=1039.055,128.362,-94.840,169.885,39.905,157.519
C08006=1039.049,128.112,-94.819,169.883,39.905,157.518
C08007=1039.043,127.863,-94.799,169.880,39.905,157.518
C08008=1039.037,127.614,-94.778,169.878,39.904,157.518
C08009=1039.031,127.365,-94.758,169.876,39.904,157.518
C08010=1039.024,127.116,-94.737,169.873,39.903,157.518
C08011=1039.018,126.866,-94.716,169.871,39.903,157.518
C08012=1039.012,126.618,-94.695,169.869,39.903,157.518
C08013=1039.005,126.369,-94.675,169.867,39.903,157.517
C08014=1039.000,126.120,-94.654,169.864,39.902,157.517
C08015=1038.993,125.871,-94.633,169.862,39.902,157.517
C08016=1038.986,125.621,-94.613,169.860,39.902,157.517
C08017=1038.979,125.336,-94.589,169.858,39.901,157.517
C08018=1038.972,125.050,-94.566,169.855,39.901,157.517
C08019=1038.965,124.764,-94.542,169.853,39.901,157.516
C08020=1038.958,124.478,-94.519,169.850,39.900,157.516
C08021=1038.952,124.229,-94.497,169.847,39.900,157.516
C08022=1038.946,123.980,-94.477,169.845,39.899,157.516
C08023=1038.939,123.731,-94.457,169.843,39.899,157.516
C08024=1038.934,123.482,-94.435,169.841,39.899,157.516
C08025=1038.927,123.233,-94.415,169.839,39.899,157.516
C08026=1038.921,122.984,-94.395,169.837,39.898,157.515
C08027=1038.915,122.735,-94.374,169.835,39.898,157.515
C08028=1038.909,122.486,-94.354,169.832,39.897,157.515
C08029=1038.902,122.236,-94.333,169.830,39.897,157.515
C08030=1038.896,121.988,-94.313,169.828,39.897,157.515
C08031=1038.890,121.738,-94.292,169.826,39.896,157.515
C08032=1038.884,121.490,-94.272,169.824,39.896,157.514
C08033=1038.878,121.240,-94.251,169.822,39.896,157.514
C08034=1038.872,120.992,-94.230,169.820,39.896,157.514
C08035=1038.865,120.742,-94.210,169.818,39.895,157.514
C08036=1038.859,120.493,-94.190,169.815,39.895,157.514
C08037=1038.853,120.244,-94.170,169.813,39.894,157.514
C08038=1038.848,119.995,-94.149,169.811,39.894,157.514
C08039=1038.841,119.746,-94.128,169.809,39.893,157.513
C08040=1038.835,119.497,-94.108,169.807,39.894,157.513
C08041=1038.829,119.248,-94.087,169.804,39.893,157.513
C08042=1038.823,118.998,-94.067,169.802,39.893,157.513
C08043=1038.817,118.749,-94.047,169.800,39.892,157.513
C08044=1038.810,118.501,-94.026,169.797,39.892,157.513
C08045=1038.805,118.251,-94.005,169.795,39.891,157.512
C08046=1038.799,118.003,-93.986,169.793,39.892,157.512
C08047=1038.792,117.753,-93.965,169.791,39.891,157.512
C08048=1038.787,117.504,-93.945,169.789,39.891,157.512
C08049=1038.780,117.254,-93.924,169.787,39.890,157.512
C08050=1038.774,117.006,-93.904,169.785,39.890,157.512
C08051=1038.768,116.757,-93.884,169.782,39.889,157.512
C08052=1038.762,116.508,-93.863,169.780,39.889,157.512
C08053=1038.756,116.259,-93.843,169.778,39.889,157.511
C08054=1038.749,116.009,-93.822,169.776,39.889,157.511
C08055=1038.743,115.761,-93.803,169.774,39.888,157.511
C08056=1038.738,115.511,-93.782,169.772,39.888,157.511
C08057=1038.732,115.262,-93.762,169.770,39.887,157.511
C08058=1038.726,115.013,-93.742,169.767,39.887,157.511
C08059=1038.720,114.764,-93.722,169.765,39.887,157.510
C08060=1038.714,114.514,-93.701,169.763,39.886,157.510
C08061=1038.708,114.266,-93.681,169.761,39.886,157.510
C08062=1038.702,114.017,-93.661,169.759,39.886,157.510
C08063=1038.695,113.767,-93.641,169.757,39.885,157.510
C08064=1038.690,113.518,-93.620,169.755,39.885,157.510
C08065=1038.684,113.269,-93.600,169.752,39.884,157.509
C08066=1038.677,113.020,-93.580,169.750,39.884,157.509
C08067=1038.671,112.771,-93.560,169.748,39.884,157.509
C08068=1038.665,112.522,-93.540,169.746,39.883,157.509
C08069=1038.659,112.273,-93.519,169.744,39.884,157.509
C08070=1038.653,112.024,-93.500,169.742,39.883,157.509
C08071=1038.646,111.774,-93.479,169.740,39.883,157.509
C08072=1038.640,111.526,-93.459,169.738,39.882,157.508
C08073=1038.634,111.277,-93.439,169.736,39.882,157.508
C08074=1038.628,111.027,-93.419,169.733,39.882,157.508
C08075=1038.622,110.778,-93.399,169.731,39.881,157.508
C08076=1038.616,110.529,-93.380,169.729,39.881,157.508
C08077=1038.609,110.279,-93.359,169.727,39.881,157.508
C08078=1038.603,110.031,-93.340,169.725,39.881,157.508
C08079=1038.597,109.782,-93.320,169.723,39.881,157.508
C08080=1038.590,109.533,-93.300,169.721,39.880,157.508
C08081=1038.583,109.247,-93.277,169.719,39.880,157.507
C08082=1038.576,108.961,-93.254,169.715,39.880,157.507
C08083=1038.569,108.675,-93.232,169.713,39.880,157.507
C08084=1038.562,108.389,-93.209,169.711,39.879,157.507
C08085=1038.555,108.140,-93.189,169.709,39.879,157.507
C08086=1038.549,107.890,-93.170,169.707,39.879,157.507
C08087=1038.543,107.641,-93.150,169.705,39.879,157.507
C08088=1038.536,107.392,-93.130,169.703,39.878,157.506
C08089=1038.530,107.143,-93.110,169.701,39.878,157.506
C08090=1038.524,106.894,-93.091,169.699,39.878,157.506
C08091=1038.518,106.645,-93.071,169.696,39.877,157.506
C08092=1038.512,106.396,-93.050,169.694,39.878,157.506
C08093=1038.506,106.146,-93.031,169.692,39.877,157.506
C08094=1038.499,105.898,-93.012,169.690,39.877,157.506
C08095=1038.493,105.648,-92.992,169.688,39.876,157.505
C08096=1038.487,105.399,-92.972,169.686,39.876,157.505
C08097=1038.481,105.150,-92.952,169.684,39.876,157.505
C08098=1038.475,104.901,-92.932,169.682,39.875,157.505
C08099=1038.468,104.651,-92.913,169.680,39.876,157.505
C08100=1038.462,104.402,-92.893,169.677,39.875,157.505
C08101=1038.456,104.154,-92.873,169.675,39.875,157.505
C08102=1038.450,103.904,-92.854,169.673,39.875,157.505
C08103=1038.444,103.655,-92.834,169.671,39.874,157.504
C08104=1038.437,103.406,-92.815,169.669,39.874,157.504
C08105=1038.431,103.157,-92.795,169.667,39.874,157.504
C08106=1038.425,102.908,-92.775,169.665,39.874,157.504
C08107=1038.420,102.659,-92.756,169.663,39.873,157.504
C08108=1038.413,102.409,-92.736,169.661,39.873,157.504
C08109=1038.406,102.161,-92.716,169.658,39.873,157.504
C08110=1038.401,101.911,-92.697,169.656,39.872,157.504
C08111=1038.395,101.662,-92.677,169.654,39.872,157.503
C08112=1038.389,101.413,-92.658,169.652,39.872,157.503
C08113=1038.382,101.163,-92.638,169.650,39.872,157.503
C08114=1038.376,100.914,-92.619,169.648,39.871,157.503
C08115=1038.370,100.665,-92.599,169.646,39.871,157.503
C08116=1038.364,100.416,-92.580,169.644,39.871,157.503
C08117=1038.358,100.167,-92.560,169.641,39.871,157.503
C08118=1038.351,99.917,-92.541,169.639,39.871,157.503
C08119=1038.345,99.669,-92.521,169.637,39.870,157.502
C08120=1038.339,99.419,-92.502,169.635,39.870,157.502
C08121=1038.333,99.171,-92.482,169.633,39.870,157.502
C08122=1038.326,98.921,-92.464,169.631,39.869,157.502
C08123=1038.320,98.671,-92.444,169.629,39.870,157.502
C08124=1038.313,98.423,-92.425,169.627,39.869,157.502
C08125=1038.308,98.173,-92.405,169.625,39.869,157.502
C08126=1038.301,97.925,-92.386,169.623,39.869,157.502
C08127=1038.295,97.675,-92.367,169.620,39.868,157.501
C08128=1038.288,97.426,-92.348,169.618,39.869,157.501
C08129=1038.282,97.177,-92.328,169.616,39.868,157.501
C08130=1038.277,96.927,-92.309,169.614,39.868,157.501
C08131=1038.270,96.678,-92.290,169.612,39.868,157.501
C08132=1038.264,96.429,-92.270,169.610,39.867,157.501
C08133=1038.258,96.180,-92.251,169.608,39.868,157.501
C08134=1038.252,95.931,-92.232,169.606,39.867,157.501
C08135=1038.245,95.682,-92.212,169.604,39.867,157.501
C08136=1038.239,95.432,-92.193,169.602,39.867,157.500
C08137=1038.233,95.183,-92.174,169.599,39.866,157.500
C08138=1038.227,94.934,-92.154,169.597,39.867,157.500
C08139=1038.220,94.685,-92.136,169.595,39.866,157.500
C08140=1038.215,94.436,-92.117,169.593,39.866,157.500
C08141=1038.208,94.187,-92.097,169.591,39.866,157.500
C08142=1038.202,93.938,-92.078,169.589,39.865,157.500
C08143=1038.195,93.688,-92.059,169.587,39.866,157.500
C08144=1038.189,93.439,-92.040,169.585,39.865,157.499
C08145=1038.183,93.154,-92.018,169.583,39.865,157.499
C08146=1038.175,92.867,-91.996,169.581,39.865,157.499
C08147=1038.168,92.582,-91.974,169.577,39.864,157.499
C08148=1038.161,92.295,-91.952,169.575,39.864,157.499
C08149=1038.155,92.046,-91.933,169.573,39.864,157.499
C08150=1038.148,91.797,-91.913,169.571,39.864,157.499
C08151=1038.143,91.548,-91.894,169.569,39.863,157.498
C08152=1038.136,91.299,-91.876,169.567,39.863,157.498
C08153=1038.131,91.049,-91.856,169.565,39.863,157.498
C08154=1038.124,90.800,-91.838,169.563,39.862,157.498
C08155=1038.118,90.551,-91.818,169.561,39.863,157.498
C08156=1038.112,90.302,-91.799,169.558,39.862,157.498
C08157=1038.106,90.052,-91.779,169.556,39.862,157.498
C08158=1038.099,89.803,-91.761,169.554,39.862,157.498
C08159=1038.093,89.554,-91.742,169.552,39.861,157.497
C08160=1038.086,89.305,-91.724,169.550,39.862,157.497
C08161=1038.080,89.056,-91.705,169.548,39.861,157.497
C08162=1038.074,88.806,-91.686,169.546,39.861,157.497
C08163=1038.068,88.557,-91.667,169.544,39.861,157.497
C08164=1038.061,88.308,-91.648,169.542,39.861,157.497
C08165=1038.055,88.059,-91.630,169.540,39.861,157.497
C08166=1038.049,87.809,-91.610,169.537,39.861,157.497
C08167=1038.043,87.560,-91.592,169.535,39.860,157.497
C08168=1038.036,87.311,-91.573,169.533,39.860,157.497
C08169=1038.030,87.062,-91.555,169.531,39.860,157.496
C08170=1038.023,86.813,-91.536,169.529,39.860,157.496
C08171=1038.018,86.563,-91.517,169.527,39.860,157.496
C08172=1038.011,86.314,-91.498,169.525,39.860,157.496
C08173=1038.005,86.065,-91.479,169.523,39.859,157.496
C08174=1037.998,85.816,-91.461,169.521,39.860,157.496
C08175=1037.992,85.567,-91.442,169.520,39.859,157.496
C08176=1037.986,85.318,-91.423,169.518,39.859,157.496
C08177=1037.980,85.068,-91.404,169.515,39.859,157.496
C08178=1037.974,84.819,-91.385,169.513,39.859,157.495
C08179=1037.967,84.570,-91.367,169.511,39.858,157.495
C08180=1037.961,84.321,-91.348,169.509,39.859,157.495
C08181=1037.955,84.072,-91.329,169.507,39.858,157.495
C08182=1037.949,83.823,-91.310,169.505,39.858,157.495
C08183=1037.942,83.573,-91.292,169.503,39.858,157.495
C08184=1037.936,83.324,-91.273,169.501,39.858,157.495
C08185=1037.930,83.075,-91.255,169.499,39.858,157.495
C08186=1037.924,82.825,-91.236,169.497,39.857,157.494
C08187=1037.917,82.576,-91.217,169.495,39.857,157.494
C08188=1037.911,82.327,-91.199,169.492,39.857,157.494
C08189=1037.905,82.078,-91.180,169.490,39.857,157.494
C08190=1037.898,81.829,-91.161,169.488,39.857,157.494
C08191=1037.892,81.580,-91.143,169.486,39.857,157.494
C08192=1037.886,81.329,-91.124,169.484,39.856,157.494
C08193=1037.880,81.080,-91.105,169.482,39.856,157.494
C08194=1037.874,80.831,-91.087,169.480,39.856,157.494
C08195=1037.867,80.582,-91.068,169.478,39.855,157.493
C08196=1037.861,80.333,-91.049,169.476,39.856,157.493
C08197=1037.855,80.085,-91.031,169.474,39.855,157.493
C08198=1037.849,79.834,-91.013,169.472,39.855,157.493
C08199=1037.843,79.585,-90.994,169.469,39.855,157.493
C08200=1037.837,79.336,-90.975,169.467,39.855,157.493
C08201=1037.830,79.087,-90.957,169.465,39.855,157.493
C08202=1037.824,78.837,-90.939,169.463,39.854,157.493
C08203=1037.818,78.588,-90.920,169.461,39.854,157.493
C08204=1037.812,78.339,-90.901,169.459,39.854,157.492
C08205=1037.806,78.090,-90.882,169.457,39.854,157.492
C08206=1037.799,77.840,-90.864,169.455,39.854,157.492
C08207=1037.794,77.592,-90.846,169.453,39.854,157.492
C08208=1037.787,77.342,-90.827,169.452,39.853,157.492
C08209=1037.779,77.056,-90.806,169.449,39.853,157.492
C08210=1037.772,76.769,-90.785,169.446,39.853,157.492
C08211=1037.765,76.484,-90.765,169.444,39.853,157.492
C08212=1037.758,76.198,-90.743,169.441,39.853,157.492
C08213=1037.752,75.949,-90.724,169.439,39.853,157.492
C08214=1037.745,75.699,-90.707,169.437,39.852,157.491
C08215=1037.739,75.451,-90.689,169.435,39.853,157.491
C08216=1037.733,75.201,-90.671,169.433,39.852,157.491
C08217=1037.726,74.952,-90.652,169.431,39.852,157.491
C08218=1037.720,74.703,-90.634,169.429,39.852,157.491
C08219=1037.714,74.453,-90.616,169.427,39.852,157.491
C08220=1037.707,74.204,-90.597,169.425,39.852,157.491
C08221=1037.701,73.954,-90.579,169.423,39.852,157.491
C08222=1037.695,73.706,-90.561,169.421,39.851,157.491
C08223=1037.689,73.456,-90.543,169.419,39.851,157.490
C08224=1037.682,73.207,-90.525,169.417,39.851,157.490
C08225=1037.676,72.958,-90.507,169.415,39.851,157.490
C08226=1037.670,72.708,-90.488,169.413,39.851,157.490
C08227=1037.664,72.459,-90.470,169.411,39.851,157.490
C08228=1037.658,72.210,-90.452,169.409,39.850,157.490
C08229=1037.651,71.961,-90.433,169.407,39.851,157.490
C08230=1037.645,71.711,-90.415,169.405,39.850,157.490
C08231=1037.639,71.462,-90.398,169.403,39.850,157.490
C08232=1037.633,71.213,-90.379,169.401,39.850,157.490
C08233=1037.626,70.964,-90.362,169.398,39.850,157.489
C08234=1037.620,70.715,-90.343,169.396,39.850,157.489
C08235=1037.614,70.465,-90.325,169.394,39.850,157.489
C08236=1037.607,70.216,-90.307,169.392,39.850,157.489
C08237=1037.601,69.966,-90.289,169.390,39.849,157.489
C08238=1037.595,69.718,-90.270,169.388,39.850,157.489
C08239=1037.589,69.468,-90.253,169.386,39.849,157.489
C08240=1037.582,69.219,-90.234,169.384,39.849,157.489
C08241=1037.576,68.969,-90.217,169.382,39.849,157.489
C08242=1037.570,68.720,-90.199,169.380,39.849,157.489
C08243=1037.563,68.472,-90.181,169.378,39.848,157.488
C08244=1037.557,68.222,-90.163,169.375,39.849,157.488
C08245=1037.551,67.972,-90.145,169.373,39.849,157.488
C08246=1037.545,67.723,-90.126,169.371,39.848,157.488
C08247=1037.538,67.474,-90.109,169.369,39.849,157.488
C08248=1037.532,67.224,-90.092,169.367,39.848,157.488
C08249=1037.526,66.975,-90.073,169.365,39.848,157.488
C08250=1037.520,66.726,-90.055,169.363,39.848,157.488
C08251=1037.514,66.477,-90.038,169.361,39.848,157.488
C08252=1037.507,66.228,-90.019,169.359,39.848,157.487
C08253=1037.501,65.978,-90.001,169.357,39.848,157.487
C08254=1037.494,65.729,-89.984,169.355,39.848,157.487
C08255=1037.489,65.480,-89.966,169.353,39.847,157.487
C08256=1037.481,65.231,-89.948,169.351,39.848,157.487
C08257=1037.475,64.981,-89.930,169.348,39.847,157.487
C08258=1037.469,64.731,-89.913,169.346,39.847,157.487
C08259=1037.463,64.482,-89.896,169.344,39.847,157.487
C08260=1037.456,64.233,-89.877,169.342,39.847,157.487
C08261=1037.450,63.984,-89.859,169.340,39.847,157.487
C08262=1037.444,63.735,-89.842,169.338,39.847,157.486
C08263=1037.438,63.485,-89.824,169.336,39.847,157.486
C08264=1037.431,63.236,-89.807,169.334,39.847,157.486
C08265=1037.425,62.987,-89.788,169.332,39.847,157.486
C08266=1037.418,62.737,-89.771,169.330,39.847,157.486
C08267=1037.412,62.488,-89.754,169.328,39.847,157.486
C08268=1037.405,62.239,-89.736,169.326,39.846,157.486
C08269=1037.399,61.989,-89.719,169.324,39.847,157.486
C08270=1037.393,61.740,-89.701,169.322,39.847,157.486
C08271=1037.386,61.491,-89.684,169.320,39.847,157.486
C08272=1037.379,61.241,-89.666,169.317,39.847,157.486
C08273=1037.372,60.955,-89.646,169.315,39.847,157.486
C08274=1037.365,60.669,-89.626,169.312,39.847,157.486
C08275=1037.358,60.383,-89.606,169.310,39.846,157.485
C08276=1037.350,60.096,-89.586,169.308,39.847,157.485
C08277=1037.343,59.847,-89.568,169.306,39.847,157.485
C08278=1037.338,59.598,-89.550,169.304,39.846,157.485
C08279=1037.331,59.349,-89.533,169.302,39.847,157.485
C08280=1037.324,59.100,-89.515,169.299,39.847,157.485
C08281=1037.318,58.850,-89.498,169.297,39.846,157.485
C08282=1037.312,58.601,-89.481,169.295,39.846,157.485
C08283=1037.305,58.352,-89.463,169.293,39.847,157.485
C08284=1037.299,58.103,-89.446,169.291,39.846,157.485
C08285=1037.292,57.853,-89.428,169.289,39.846,157.485
C08286=1037.285,57.604,-89.411,169.287,39.847,157.485
C08287=1037.280,57.355,-89.393,169.284,39.846,157.484
C08288=1037.273,57.105,-89.376,169.282,39.846,157.484
C08289=1037.267,56.855,-89.359,169.280,39.846,157.484
C08290=1037.261,56.606,-89.342,169.278,39.846,157.484
C08291=1037.254,56.357,-89.325,169.276,39.846,157.484
C08292=1037.249,56.108,-89.307,169.274,39.846,157.484
C08293=1037.242,55.858,-89.290,169.272,39.846,157.484
C08294=1037.235,55.609,-89.272,169.270,39.846,157.484
C08295=1037.229,55.360,-89.255,169.268,39.846,157.484
C08296=1037.223,55.110,-89.237,169.266,39.846,157.484
C08297=1037.216,54.862,-89.220,169.264,39.846,157.484
C08298=1037.210,54.612,-89.202,169.262,39.846,157.483
C08299=1037.203,54.362,-89.185,169.260,39.846,157.483
C08300=1037.197,54.114,-89.168,169.258,39.846,157.483
C08301=1037.191,53.863,-89.151,169.256,39.846,157.483
C08302=1037.185,53.615,-89.134,169.253,39.845,157.483
C08303=1037.178,53.365,-89.117,169.251,39.846,157.483
C08304=1037.172,53.115,-89.099,169.249,39.845,157.483
C08305=1037.166,52.867,-89.082,169.247,39.845,157.483
C08306=1037.159,52.617,-89.064,169.245,39.846,157.483
C08307=1037.153,52.368,-89.047,169.243,39.845,157.483
C08308=1037.147,52.118,-89.030,169.241,39.845,157.483
C08309=1037.141,51.869,-89.013,169.239,39.845,157.483
C08310=1037.134,51.620,-88.995,169.237,39.845,157.482
C08311=1037.128,51.371,-88.978,169.235,39.845,157.482
C08312=1037.121,51.122,-88.961,169.233,39.845,157.482
C08313=1037.116,50.872,-88.944,169.231,39.845,157.482
C08314=1037.109,50.622,-88.927,169.229,39.845,157.482
C08315=1037.103,50.374,-88.910,169.227,39.845,157.482
C08316=1037.097,50.124,-88.892,169.224,39.845,157.482
C08317=1037.091,49.875,-88.876,169.222,39.845,157.482
C08318=1037.084,49.625,-88.858,169.220,39.844,157.482
C08319=1037.079,49.376,-88.841,169.218,39.845,157.482
C08320=1037.072,49.127,-88.823,169.216,39.844,157.481
C08321=1037.066,48.877,-88.807,169.214,39.844,157.481
C08322=1037.060,48.628,-88.789,169.212,39.844,157.481
C08323=1037.053,48.379,-88.772,169.210,39.844,157.481
C08324=1037.047,48.130,-88.755,169.208,39.844,157.481
C08325=1037.041,47.880,-88.739,169.206,39.844,157.481
C08326=1037.034,47.630,-88.721,169.204,39.844,157.481
C08327=1037.028,47.382,-88.704,169.202,39.843,157.481
C08328=1037.022,47.132,-88.687,169.200,39.844,157.481
C08329=1037.016,46.883,-88.670,169.198,39.844,157.481
C08330=1037.009,46.633,-88.652,169.195,39.843,157.480
C08331=1037.003,46.384,-88.636,169.193,39.843,157.480
C08332=1036.998,46.135,-88.618,169.191,39.843,157.480
C08333=1036.991,45.885,-88.601,169.189,39.843,157.480
C08334=1036.985,45.636,-88.585,169.187,39.843,157.480
C08335=1036.978,45.387,-88.567,169.185,39.843,157.480
C08336=1036.973,45.138,-88.550,169.183,39.843,157.480
C08337=1036.963,44.769,-88.525,169.180,39.843,157.480
C08338=1036.955,44.401,-88.500,169.177,39.842,157.480
C08339=1036.945,44.033,-88.475,169.174,39.843,157.479
C08340=1036.935,43.665,-88.450,169.170,39.842,157.479
C08341=1036.930,43.415,-88.433,169.168,39.842,157.479
C08342=1036.924,43.167,-88.416,169.166,39.842,157.479
C08343=1036.917,42.917,-88.399,169.164,39.842,157.479
C08344=1036.911,42.668,-88.382,169.162,39.842,157.479
C08345=1036.905,42.418,-88.366,169.160,39.842,157.479
C08346=1036.898,42.169,-88.349,169.158,39.842,157.479
C08347=1036.892,41.920,-88.333,169.156,39.842,157.479
C08348=1036.886,41.670,-88.315,169.154,39.842,157.479
C08349=1036.880,41.421,-88.299,169.152,39.842,157.479
C08350=1036.873,41.172,-88.282,169.150,39.842,157.478
C08351=1036.867,40.922,-88.265,169.148,39.841,157.478
C08352=1036.861,40.673,-88.249,169.146,39.842,157.478
C08353=1036.854,40.423,-88.232,169.144,39.842,157.478
C08354=1036.848,40.174,-88.216,169.140,39.841,157.478
C08355=1036.841,39.925,-88.198,169.138,39.842,157.478
C08356=1036.835,39.675,-88.182,169.136,39.842,157.478
C08357=1036.829,39.427,-88.165,169.134,39.841,157.478
C08358=1036.822,39.176,-88.148,169.132,39.841,157.478
C08359=1036.816,38.927,-88.132,169.130,39.842,157.478
C08360=1036.810,38.678,-88.115,169.128,39.841,157.478
C08361=1036.804,38.428,-88.098,169.126,39.841,157.477
C08362=1036.798,38.179,-88.082,169.124,39.842,157.477
C08363=1036.791,37.930,-88.065,169.122,39.841,157.477
C08364=1036.785,37.680,-88.049,169.120,39.841,157.477
C08365=1036.779,37.431,-88.032,169.118,39.841,157.477
C08366=1036.773,37.182,-88.015,169.116,39.842,157.477
C08367=1036.766,36.932,-87.999,169.114,39.841,157.477
C08368=1036.760,36.683,-87.983,169.112,39.841,157.477
C08369=1036.754,36.434,-87.966,169.110,39.841,157.477
C08370=1036.747,36.184,-87.950,169.108,39.842,157.477
C08371=1036.741,35.935,-87.933,169.105,39.841,157.477
C08372=1036.735,35.686,-87.917,169.102,39.841,157.477
C08373=1036.728,35.436,-87.900,169.100,39.842,157.477
C08374=1036.722,35.187,-87.883,169.098,39.842,157.477
C08375=1036.715,34.938,-87.868,169.096,39.842,157.476
C08376=1036.709,34.688,-87.851,169.094,39.841,157.476
C08377=1036.703,34.438,-87.835,169.092,39.842,157.476
C08378=1036.696,34.190,-87.818,169.090,39.842,157.476
C08379=1036.690,33.940,-87.801,169.088,39.842,157.476
C08380=1036.683,33.691,-87.786,169.086,39.841,157.476
C08381=1036.677,33.441,-87.769,169.084,39.842,157.476
C08382=1036.671,33.191,-87.753,169.082,39.842,157.476
C08383=1036.665,32.942,-87.736,169.080,39.842,157.476
C08384=1036.658,32.693,-87.720,169.078,39.842,157.476
C08385=1036.652,32.444,-87.704,169.075,39.842,157.476
C08386=1036.645,32.194,-87.687,169.073,39.842,157.476
C08387=1036.639,31.945,-87.671,169.071,39.842,157.476
C08388=1036.633,31.695,-87.655,169.069,39.842,157.475
C08389=1036.627,31.446,-87.639,169.067,39.842,157.475
C08390=1036.620,31.196,-87.622,169.065,39.842,157.475
C08391=1036.614,30.947,-87.606,169.063,39.842,157.475
C08392=1036.608,30.698,-87.590,169.060,39.842,157.475
C08393=1036.601,30.449,-87.574,169.058,39.842,157.475
C08394=1036.595,30.199,-87.557,169.056,39.842,157.475
C08395=1036.589,29.950,-87.541,169.054,39.842,157.475
C08396=1036.583,29.700,-87.524,169.052,39.842,157.475
C08397=1036.574,29.365,-87.503,169.049,39.842,157.475
C08398=1036.566,29.029,-87.481,169.046,39.842,157.475
C08399=1036.558,28.743,-87.462,169.044,39.842,157.474
C08400=1036.552,28.456,-87.444,169.041,39.842,157.474
C08401=1036.544,28.169,-87.425,169.039,39.842,157.474
C08402=1036.536,27.882,-87.406,169.036,39.843,157.474
C08403=1036.530,27.633,-87.391,169.034,39.842,157.474
C08404=1036.524,27.383,-87.375,169.032,39.842,157.474
C08405=1036.518,27.134,-87.359,169.030,39.842,157.474
C08406=1036.511,26.884,-87.343,169.028,39.843,157.474
C08407=1036.505,26.635,-87.327,169.026,39.843,157.474
C08408=1036.498,26.386,-87.311,169.023,39.842,157.474
C08409=1036.492,26.137,-87.295,169.021,39.842,157.474
C08410=1036.486,25.888,-87.279,169.019,39.843,157.474
C08411=1036.479,25.637,-87.262,169.016,39.843,157.474
C08412=1036.473,25.388,-87.246,169.014,39.843,157.474
C08413=1036.466,25.139,-87.230,169.012,39.843,157.474
C08414=1036.460,24.890,-87.214,169.010,39.843,157.473
C08415=1036.454,24.640,-87.199,169.008,39.843,157.473
C08416=1036.448,24.391,-87.183,169.006,39.843,157.473
C08417=1036.441,24.141,-87.167,169.004,39.843,157.473
C08418=1036.435,23.892,-87.151,169.002,39.843,157.473
C08419=1036.428,23.643,-87.135,168.999,39.844,157.473
C08420=1036.422,23.393,-87.119,168.997,39.843,157.473
C08421=1036.416,23.144,-87.104,168.995,39.843,157.473
C08422=1036.410,22.894,-87.088,168.993,39.844,157.473
C08423=1036.403,22.645,-87.072,168.991,39.844,157.473
C08424=1036.397,22.395,-87.055,168.989,39.844,157.473
C08425=1036.390,22.146,-87.040,168.987,39.843,157.473
C08426=1036.384,21.896,-87.024,168.985,39.844,157.473
C08427=1036.378,21.647,-87.008,168.982,39.844,157.472
C08428=1036.372,21.398,-86.992,168.980,39.844,157.472
C08429=1036.365,21.149,-86.977,168.978,39.844,157.472
C08430=1036.359,20.899,-86.961,168.975,39.844,157.472
C08431=1036.353,20.650,-86.945,168.973,39.844,157.472
C08432=1036.347,20.400,-86.929,168.971,39.844,157.472
C08433=1036.339,20.151,-86.913,168.969,39.844,157.472
C08434=1036.334,19.901,-86.897,168.967,39.844,157.472
C08435=1036.327,19.652,-86.882,168.964,39.844,157.472
C08436=1036.321,19.402,-86.866,168.962,39.844,157.472
C08437=1036.315,19.153,-86.851,168.960,39.844,157.472
C08438=1036.308,18.904,-86.835,168.958,39.845,157.472
C08439=1036.302,18.654,-86.819,168.956,39.845,157.472
C08440=1036.296,18.405,-86.804,168.954,39.845,157.472
C08441=1036.290,18.155,-86.788,168.952,39.845,157.472
C08442=1036.283,17.906,-86.772,168.949,39.845,157.472
C08443=1036.277,17.657,-86.757,168.947,39.845,157.471
C08444=1036.271,17.407,-86.741,168.945,39.845,157.471
C08445=1036.264,17.157,-86.725,168.943,39.845,157.471
C08446=1036.257,16.908,-86.710,168.941,39.845,157.471
C08447=1036.251,16.658,-86.693,168.939,39.846,157.471
C08448=1036.245,16.409,-86.678,168.937,39.846,157.471
C08449=1036.238,16.160,-86.663,168.934,39.846,157.471
C08450=1036.232,15.910,-86.647,168.932,39.846,157.471
C08451=1036.226,15.661,-86.632,168.930,39.846,157.471
C08452=1036.219,15.411,-86.617,168.928,39.846,157.471
C08453=1036.213,15.162,-86.600,168.926,39.846,157.471
C08454=1036.207,14.913,-86.585,168.923,39.846,157.471
C08455=1036.200,14.663,-86.570,168.920,39.846,157.471
C08456=1036.194,14.414,-86.554,168.918,39.847,157.471
C08457=1036.188,14.164,-86.539,168.916,39.846,157.470
C08458=1036.181,13.915,-86.523,168.914,39.846,157.470
C08459=1036.176,13.665,-86.507,168.912,39.847,157.470
C08460=1036.169,13.415,-86.492,168.910,39.847,157.470
C08461=1036.163,13.166,-86.477,168.907,39.847,157.470
C08462=1036.156,12.917,-86.462,168.905,39.847,157.470
C08463=1036.149,12.631,-86.444,168.903,39.847,157.470
C08464=1036.141,12.346,-86.426,168.900,39.848,157.470
C08465=1036.134,12.061,-86.409,168.898,39.848,157.470
C08466=1036.126,11.775,-86.392,168.895,39.848,157.470
C08467=1036.120,11.526,-86.376,168.893,39.848,157.470
C08468=1036.113,11.277,-86.361,168.891,39.848,157.470
C08469=1036.107,11.027,-86.346,168.889,39.849,157.470
C08470=1036.100,10.778,-86.331,168.886,39.849,157.470
C08471=1036.094,10.528,-86.316,168.884,39.849,157.470
C08472=1036.088,10.278,-86.300,168.882,39.849,157.470
C08473=1036.082,10.029,-86.284,168.880,39.849,157.470
C08474=1036.075,9.779,-86.270,168.877,39.850,157.470
C08475=1036.069,9.530,-86.255,168.875,39.850,157.470
C08476=1036.062,9.281,-86.239,168.873,39.850,157.469
C08477=1036.056,9.032,-86.224,168.871,39.850,157.469
C08478=1036.050,8.782,-86.209,168.869,39.850,157.469
C08479=1036.043,8.533,-86.194,168.866,39.851,157.469
C08480=1036.037,8.284,-86.179,168.864,39.851,157.469
C08481=1036.030,8.034,-86.164,168.862,39.851,157.469
C08482=1036.024,7.784,-86.149,168.860,39.851,157.469
C08483=1036.017,7.535,-86.133,168.858,39.851,157.469
C08484=1036.011,7.285,-86.118,168.855,39.852,157.469
C08485=1036.005,7.036,-86.103,168.853,39.852,157.469
C08486=1035.999,6.786,-86.088,168.851,39.852,157.469
C08487=1035.992,6.537,-86.072,168.849,39.852,157.469
C08488=1035.986,6.287,-86.057,168.846,39.852,157.469
C08489=1035.980,6.038,-86.043,168.843,39.852,157.469
C08490=1035.974,5.789,-86.028,168.841,39.852,157.469
C08491=1035.967,5.539,-86.013,168.839,39.852,157.469
C08492=1035.961,5.290,-85.997,168.837,39.852,157.469
C08493=1035.954,5.040,-85.982,168.834,39.853,157.469
C08494=1035.948,4.791,-85.967,168.832,39.853,157.468
C08495=1035.941,4.541,-85.952,168.830,39.853,157.468
C08496=1035.935,4.291,-85.937,168.828,39.853,157.468
C08497=1035.929,4.042,-85.923,168.826,39.853,157.468
C08498=1035.923,3.793,-85.907,168.823,39.854,157.468
C08499=1035.916,3.544,-85.892,168.821,39.854,157.468
C08500=1035.910,3.294,-85.877,168.819,39.854,157.468
C08501=1035.903,3.044,-85.862,168.817,39.854,157.468
C08502=1035.897,2.795,-85.847,168.815,39.854,157.468
C08503=1035.891,2.546,-85.833,168.812,39.855,157.468
C08504=1035.885,2.296,-85.818,168.810,39.855,157.468
C08505=1035.879,2.046,-85.803,168.808,39.854,157.468
C08506=1035.872,1.797,-85.787,168.806,39.854,157.468
C08507=1035.865,1.548,-85.772,168.803,39.855,157.468
C08508=1035.860,1.299,-85.758,168.801,39.855,157.468
C08509=1035.853,1.049,-85.743,168.799,39.855,157.468
C08510=1035.847,0.799,-85.728,168.797,39.855,157.468
C08511=1035.841,0.550,-85.713,168.795,39.855,157.468
C08512=1035.834,0.300,-85.698,168.792,39.856,157.467
C08513=1035.828,0.051,-85.683,168.790,39.856,157.467
C08514=1035.822,-0.199,-85.668,168.788,39.856,157.467
C08515=1035.816,-0.448,-85.653,168.786,39.856,157.467
C08516=1035.810,-0.698,-85.638,168.783,39.856,157.467
C08517=1035.804,-0.947,-85.623,168.780,39.856,157.467
C08518=1035.798,-1.197,-85.608,168.778,39.856,157.467
C08519=1035.791,-1.446,-85.593,168.776,39.856,157.467
C08520=1035.785,-1.696,-85.578,168.773,39.857,157.467
C08521=1035.779,-1.945,-85.564,168.771,39.857,157.467
C08522=1035.773,-2.195,-85.549,168.769,39.857,157.467
C08523=1035.766,-2.444,-85.534,168.767,39.857,157.467
C08524=1035.761,-2.693,-85.519,168.765,39.857,157.467
C08525=1035.754,-2.943,-85.504,168.762,39.857,157.467
C08526=1035.748,-3.193,-85.489,168.760,39.858,157.467
C08527=1035.741,-3.476,-85.473,168.758,39.857,157.466
C08528=1035.734,-3.760,-85.457,168.755,39.857,157.466
C08529=1035.727,-4.043,-85.440,168.752,39.858,157.466
C08530=1035.719,-4.326,-85.423,168.750,39.859,157.466
C08531=1035.713,-4.576,-85.409,168.747,39.859,157.466
C08532=1035.706,-4.826,-85.395,168.745,39.859,157.466
C08533=1035.700,-5.075,-85.380,168.743,39.859,157.466
C08534=1035.694,-5.324,-85.365,168.741,39.859,157.466
C08535=1035.687,-5.573,-85.351,168.738,39.860,157.466
C08536=1035.681,-5.824,-85.337,168.736,39.860,157.466
C08537=1035.675,-6.073,-85.322,168.734,39.860,157.466
C08538=1035.668,-6.322,-85.308,168.731,39.860,157.466
C08539=1035.661,-6.572,-85.293,168.729,39.861,157.466
C08540=1035.655,-6.822,-85.278,168.727,39.861,157.466
C08541=1035.649,-7.071,-85.265,168.724,39.861,157.466
C08542=1035.642,-7.320,-85.250,168.722,39.862,157.466
C08543=1035.636,-7.570,-85.235,168.720,39.862,157.466
C08544=1035.630,-7.819,-85.221,168.718,39.862,157.466
C08545=1035.624,-8.069,-85.206,168.715,39.862,157.466
C08546=1035.617,-8.319,-85.191,168.713,39.862,157.466
C08547=1035.611,-8.568,-85.178,168.711,39.863,157.466
C08548=1035.605,-8.817,-85.163,168.708,39.863,157.466
C08549=1035.598,-9.067,-85.148,168.706,39.863,157.466
C08550=1035.592,-9.316,-85.135,168.704,39.864,157.466
C08551=1035.586,-9.566,-85.120,168.701,39.864,157.466
C08552=1035.578,-9.815,-85.106,168.699,39.864,157.465
C08553=1035.573,-10.065,-85.092,168.697,39.864,157.465
C08554=1035.567,-10.315,-85.077,168.694,39.865,157.465
C08555=1035.560,-10.563,-85.063,168.692,39.865,157.465
C08556=1035.554,-10.814,-85.049,168.690,39.865,157.465
C08557=1035.548,-11.063,-85.034,168.688,39.865,157.465
C08558=1035.541,-11.312,-85.020,168.685,39.865,157.465
C08559=1035.535,-11.562,-85.006,168.683,39.866,157.465
C08560=1035.529,-11.812,-84.991,168.681,39.866,157.465
C08561=1035.522,-12.061,-84.977,168.678,39.866,157.465
C08562=1035.516,-12.311,-84.962,168.676,39.866,157.465
C08563=1035.510,-12.560,-84.949,168.674,39.867,157.465
C08564=1035.503,-12.810,-84.934,168.671,39.867,157.465
C08565=1035.498,-13.059,-84.920,168.669,39.868,157.465
C08566=1035.491,-13.309,-84.906,168.667,39.868,157.465
C08567=1035.484,-13.558,-84.891,168.664,39.868,157.465
C08568=1035.479,-13.808,-84.877,168.662,39.868,157.465
C08569=1035.472,-14.057,-84.863,168.660,39.868,157.465
C08570=1035.466,-14.307,-84.849,168.657,39.869,157.465
C08571=1035.459,-14.556,-84.835,168.655,39.869,157.465
C08572=1035.454,-14.806,-84.821,168.653,39.869,157.465
C08573=1035.447,-15.055,-84.806,168.650,39.869,157.465
C08574=1035.441,-15.305,-84.792,168.647,39.869,157.464
C08575=1035.435,-15.555,-84.778,168.645,39.870,157.464
C08576=1035.429,-15.803,-84.764,168.643,39.870,157.464
C08577=1035.422,-16.054,-84.750,168.641,39.871,157.464
C08578=1035.415,-16.303,-84.736,168.639,39.871,157.464
C08579=1035.409,-16.552,-84.722,168.635,39.871,157.464
C08580=1035.403,-16.803,-84.708,168.633,39.871,157.464
C08581=1035.397,-17.051,-84.694,168.631,39.872,157.464
C08582=1035.390,-17.301,-84.681,168.629,39.872,157.464
C08583=1035.384,-17.551,-84.667,168.627,39.873,157.464
C08584=1035.377,-17.800,-84.652,168.624,39.873,157.464
C08585=1035.372,-18.050,-84.638,168.621,39.873,157.464
C08586=1035.365,-18.300,-84.625,168.620,39.874,157.464
C08587=1035.358,-18.548,-84.611,168.617,39.874,157.464
C08588=1035.352,-18.799,-84.597,168.615,39.874,157.464
C08589=1035.346,-19.048,-84.583,168.612,39.874,157.464
C08590=1035.339,-19.297,-84.569,168.609,39.875,157.464
C08591=1035.332,-19.579,-84.554,168.607,39.876,157.464
C08592=1035.325,-19.861,-84.538,168.605,39.876,157.464
C08593=1035.318,-20.143,-84.523,168.602,39.876,157.464
C08594=1035.311,-20.424,-84.507,168.599,39.876,157.464
C08595=1035.305,-20.674,-84.493,168.597,39.877,157.464
C08596=1035.298,-20.924,-84.479,168.595,39.877,157.464
C08597=1035.292,-21.173,-84.465,168.592,39.878,157.464
C08598=1035.286,-21.423,-84.451,168.590,39.878,157.464
C08599=1035.280,-21.672,-84.438,168.587,39.878,157.464
C08600=1035.273,-21.922,-84.424,168.585,39.879,157.464
C08601=1035.267,-22.171,-84.410,168.583,39.879,157.464
C08602=1035.260,-22.421,-84.396,168.580,39.879,157.464
C08603=1035.254,-22.670,-84.383,168.578,39.879,157.464
C08604=1035.248,-22.920,-84.369,168.575,39.880,157.464
C08605=1035.242,-23.170,-84.355,168.572,39.880,157.463
C08606=1035.235,-23.419,-84.342,168.571,39.881,157.464
C08607=1035.229,-23.669,-84.327,168.568,39.881,157.463
C08608=1035.223,-23.918,-84.314,168.566,39.881,157.463
C08609=1035.217,-24.167,-84.300,168.563,39.881,157.463
C08610=1035.211,-24.417,-84.286,168.561,39.882,157.463
C08611=1035.204,-24.667,-84.273,168.559,39.882,157.463
C08612=1035.198,-24.916,-84.260,168.556,39.883,157.463
C08613=1035.192,-25.166,-84.245,168.554,39.883,157.463
C08614=1035.185,-25.415,-84.231,168.551,39.883,157.463
C08615=1035.179,-25.665,-84.218,168.549,39.883,157.463
C08616=1035.173,-25.914,-84.204,168.546,39.883,157.463
C08617=1035.167,-26.164,-84.191,168.544,39.884,157.463
C08618=1035.160,-26.414,-84.177,168.542,39.885,157.463
C08619=1035.155,-26.663,-84.163,168.539,39.885,157.463
C08620=1035.148,-26.913,-84.150,168.537,39.885,157.463
C08621=1035.142,-27.162,-84.136,168.534,39.885,157.463
C08622=1035.135,-27.412,-84.123,168.532,39.886,157.463
C08623=1035.129,-27.661,-84.110,168.530,39.886,157.463
C08624=1035.122,-27.911,-84.096,168.527,39.886,157.463
C08625=1035.116,-28.160,-84.083,168.525,39.887,157.463
C08626=1035.111,-28.410,-84.069,168.522,39.888,157.463
C08627=1035.104,-28.660,-84.055,168.520,39.888,157.463
C08628=1035.098,-28.909,-84.042,168.517,39.889,157.463
C08629=1035.091,-29.158,-84.029,168.515,39.889,157.463
C08630=1035.085,-29.409,-84.016,168.512,39.889,157.463
C08631=1035.079,-29.658,-84.003,168.510,39.890,157.463
C08632=1035.073,-29.907,-83.989,168.508,39.890,157.463
C08633=1035.066,-30.157,-83.976,168.505,39.890,157.463
C08634=1035.060,-30.407,-83.962,168.503,39.891,157.463
C08635=1035.053,-30.656,-83.949,168.500,39.891,157.463
C08636=1035.046,-30.906,-83.935,168.498,39.892,157.463
C08637=1035.040,-31.155,-83.922,168.495,39.893,157.463
C08638=1035.034,-31.405,-83.910,168.493,39.893,157.463
C08639=1035.028,-31.654,-83.896,168.490,39.893,157.463
C08640=1035.021,-31.904,-83.883,168.488,39.894,157.463
C08641=1035.015,-32.154,-83.869,168.485,39.894,157.463
C08642=1035.009,-32.403,-83.856,168.483,39.894,157.463
C08643=1035.002,-32.653,-83.843,168.480,39.895,157.463
C08644=1034.996,-32.903,-83.830,168.478,39.895,157.463
C08645=1034.990,-33.152,-83.817,168.475,39.896,157.463
C08646=1034.984,-33.401,-83.803,168.473,39.896,157.463
C08647=1034.978,-33.651,-83.790,168.471,39.897,157.463
C08648=1034.971,-33.901,-83.776,168.468,39.897,157.463
C08649=1034.966,-34.151,-83.763,168.466,39.898,157.463
C08650=1034.959,-34.400,-83.750,168.463,39.898,157.463
C08651=1034.953,-34.649,-83.737,168.461,39.898,157.463
C08652=1034.946,-34.899,-83.723,168.458,39.899,157.463
C08653=1034.940,-35.149,-83.711,168.456,39.899,157.463
C08654=1034.934,-35.398,-83.697,168.453,39.900,157.462
C08655=1034.927,-35.680,-83.683,168.450,39.900,157.462
C08656=1034.920,-35.960,-83.668,168.448,39.901,157.462
C08657=1034.913,-36.241,-83.653,168.445,39.902,157.463
C08658=1034.905,-36.522,-83.638,168.442,39.902,157.462
C08659=1034.900,-36.772,-83.626,168.440,39.902,157.462
C08660=1034.893,-37.021,-83.612,168.437,39.903,157.462
C08661=1034.887,-37.271,-83.599,168.435,39.903,157.462
C08662=1034.881,-37.521,-83.586,168.432,39.903,157.462
C08663=1034.875,-37.770,-83.573,168.430,39.904,157.462
C08664=1034.869,-38.019,-83.560,168.427,39.904,157.462
C08665=1034.862,-38.270,-83.547,168.425,39.905,157.462
C08666=1034.856,-38.519,-83.534,168.422,39.905,157.462
C08667=1034.850,-38.769,-83.521,168.420,39.906,157.462
C08668=1034.844,-39.018,-83.508,168.417,39.906,157.462
C08669=1034.838,-39.268,-83.495,168.415,39.907,157.462
C08670=1034.832,-39.517,-83.482,168.412,39.907,157.462
C08671=1034.825,-39.767,-83.470,168.410,39.908,157.462
C08672=1034.818,-40.017,-83.456,168.408,39.908,157.462
C08673=1034.812,-40.266,-83.443,168.405,39.909,157.462
C08674=1034.806,-40.516,-83.431,168.403,39.909,157.462
C08675=1034.799,-40.765,-83.418,168.400,39.910,157.462
C08676=1034.793,-41.015,-83.405,168.398,39.910,157.462
C08677=1034.787,-41.265,-83.393,168.395,39.911,157.462
C08678=1034.781,-41.514,-83.380,168.393,39.912,157.462
C08679=1034.775,-41.763,-83.368,168.390,39.912,157.462
C08680=1034.768,-42.013,-83.354,168.388,39.913,157.462
C08681=1034.762,-42.263,-83.341,168.385,39.913,157.462
C08682=1034.756,-42.513,-83.328,168.382,39.914,157.462
C08683=1034.749,-42.762,-83.316,168.380,39.914,157.462
C08684=1034.743,-43.011,-83.303,168.377,39.915,157.462
C08685=1034.737,-43.261,-83.290,168.375,39.915,157.462
C08686=1034.731,-43.511,-83.278,168.372,39.916,157.462
C08687=1034.724,-43.760,-83.265,168.370,39.916,157.462
C08688=1034.718,-44.010,-83.253,168.367,39.917,157.462
C08689=1034.712,-44.259,-83.239,168.365,39.917,157.462
C08690=1034.705,-44.509,-83.227,168.362,39.918,157.462
C08691=1034.699,-44.759,-83.215,168.360,39.918,157.462
C08692=1034.693,-45.008,-83.202,168.357,39.919,157.462
C08693=1034.687,-45.258,-83.189,168.354,39.920,157.462
C08694=1034.681,-45.507,-83.177,168.352,39.920,157.462
C08695=1034.674,-45.757,-83.164,168.349,39.921,157.462
C08696=1034.668,-46.007,-83.151,168.347,39.922,157.462
C08697=1034.662,-46.256,-83.139,168.344,39.922,157.462
C08698=1034.656,-46.505,-83.126,168.343,39.923,157.462
C08699=1034.650,-46.755,-83.113,168.340,39.923,157.462
C08700=1034.644,-47.005,-83.101,168.337,39.924,157.462
C08701=1034.637,-47.255,-83.089,168.335,39.924,157.462
C08702=1034.631,-47.504,-83.076,168.332,39.925,157.462
C08703=1034.625,-47.754,-83.063,168.330,39.925,157.462
C08704=1034.618,-48.003,-83.051,168.327,39.926,157.462
C08705=1034.612,-48.253,-83.039,168.325,39.926,157.462
C08706=1034.606,-48.503,-83.025,168.322,39.926,157.462
C08707=1034.600,-48.753,-83.013,168.320,39.927,157.462
C08708=1034.594,-49.002,-83.001,168.317,39.928,157.462
C08709=1034.588,-49.252,-82.988,168.314,39.928,157.462
C08710=1034.582,-49.501,-82.975,168.312,39.929,157.462
C08711=1034.575,-49.751,-82.963,168.309,39.930,157.462
C08712=1034.569,-50.001,-82.950,168.307,39.930,157.462
C08713=1034.563,-50.251,-82.938,168.304,39.931,157.462
C08714=1034.556,-50.500,-82.926,168.302,39.931,157.462
C08715=1034.551,-50.749,-82.914,168.299,39.932,157.462
C08716=1034.544,-50.998,-82.901,168.296,39.933,157.462
C08717=1034.538,-51.248,-82.889,168.294,39.933,157.462
C08718=1034.532,-51.498,-82.877,168.291,39.934,157.462
C08719=1034.525,-51.780,-82.863,168.288,39.935,157.462
C08720=1034.517,-52.062,-82.850,168.286,39.936,157.462
C08721=1034.510,-52.342,-82.836,168.283,39.937,157.462
C08722=1034.503,-52.624,-82.822,168.280,39.937,157.462
C08723=1034.496,-52.874,-82.810,168.277,39.938,157.462
C08724=1034.490,-53.123,-82.798,168.275,39.939,157.462
C08725=1034.484,-53.373,-82.785,168.272,39.940,157.463
C08726=1034.477,-53.623,-82.774,168.269,39.940,157.462
C08727=1034.471,-53.872,-82.762,168.267,39.941,157.463
C08728=1034.465,-54.122,-82.749,168.264,39.942,157.463
C08729=1034.459,-54.371,-82.737,168.261,39.942,157.463
C08730=1034.452,-54.621,-82.725,168.259,39.943,157.463
C08731=1034.446,-54.871,-82.713,168.256,39.944,157.463
C08732=1034.439,-55.120,-82.701,168.254,39.944,157.463
C08733=1034.433,-55.370,-82.689,168.251,39.945,157.463
C08734=1034.427,-55.620,-82.676,168.248,39.946,157.463
C08735=1034.420,-55.869,-82.664,168.247,39.946,157.463
C08736=1034.414,-56.118,-82.653,168.244,39.947,157.463
C08737=1034.408,-56.368,-82.640,168.241,39.948,157.463
C08738=1034.402,-56.618,-82.629,168.239,39.949,157.463
C08739=1034.395,-56.868,-82.617,168.236,39.949,157.463
C08740=1034.389,-57.117,-82.605,168.233,39.950,157.463
C08741=1034.383,-57.367,-82.593,168.231,39.951,157.463
C08742=1034.377,-57.616,-82.581,168.228,39.951,157.463
C08743=1034.370,-57.866,-82.569,168.225,39.952,157.463
C08744=1034.364,-58.116,-82.557,168.223,39.953,157.463
C08745=1034.358,-58.366,-82.545,168.220,39.954,157.463
C08746=1034.351,-58.615,-82.533,168.217,39.954,157.463
C08747=1034.345,-58.865,-82.521,168.215,39.955,157.463
C08748=1034.339,-59.114,-82.509,168.212,39.956,157.463
C08749=1034.332,-59.364,-82.497,168.210,39.957,157.463
C08750=1034.326,-59.614,-82.486,168.208,39.957,157.463
C08751=1034.320,-59.864,-82.473,168.205,39.958,157.463
C08752=1034.314,-60.113,-82.462,168.202,39.959,157.463
C08753=1034.308,-60.362,-82.450,168.200,39.959,157.463
C08754=1034.302,-60.613,-82.438,168.197,39.960,157.463
C08755=1034.295,-60.862,-82.426,168.194,39.961,157.463
C08756=1034.289,-61.111,-82.414,168.191,39.962,157.463
C08757=1034.283,-61.361,-82.402,168.189,39.962,157.463
C08758=1034.277,-61.611,-82.391,168.186,39.963,157.463
C08759=1034.270,-61.861,-82.379,168.183,39.964,157.463
C08760=1034.264,-62.110,-82.367,168.181,39.964,157.463
C08761=1034.258,-62.360,-82.356,168.178,39.965,157.463
C08762=1034.252,-62.610,-82.343,168.175,39.966,157.463
C08763=1034.246,-62.859,-82.332,168.173,39.966,157.463
C08764=1034.239,-63.108,-82.320,168.171,39.967,157.463
C08765=1034.233,-63.358,-82.309,168.168,39.968,157.464
C08766=1034.228,-63.608,-82.296,168.166,39.969,157.464
C08767=1034.221,-63.858,-82.285,168.163,39.969,157.464
C08768=1034.215,-64.107,-82.273,168.160,39.970,157.464
C08769=1034.209,-64.356,-82.262,168.158,39.971,157.464
C08770=1034.203,-64.607,-82.250,168.155,39.972,157.464
C08771=1034.196,-64.856,-82.238,168.152,39.972,157.464
C08772=1034.190,-65.105,-82.226,168.150,39.973,157.464
C08773=1034.184,-65.355,-82.215,168.147,39.974,157.464
C08774=1034.178,-65.605,-82.202,168.144,39.975,157.464
C08775=1034.172,-65.855,-82.191,168.141,39.975,157.464
C08776=1034.166,-66.104,-82.180,168.139,39.976,157.464
C08777=1034.159,-66.354,-82.168,168.137,39.977,157.464
C08778=1034.154,-66.604,-82.156,168.134,39.978,157.464
C08779=1034.147,-66.853,-82.144,168.132,39.978,157.464
C08780=1034.142,-67.103,-82.133,168.129,39.979,157.464
C08781=1034.135,-67.352,-82.121,168.126,39.980,157.464
C08782=1034.129,-67.602,-82.110,168.124,39.981,157.464
C08783=1034.122,-67.885,-82.097,168.121,39.981,157.464
C08784=1034.115,-68.168,-82.084,168.118,39.982,157.464
C08785=1034.109,-68.450,-82.071,168.114,39.983,157.464
C08786=1034.102,-68.733,-82.058,168.111,39.984,157.464
C08787=1034.096,-68.983,-82.045,168.109,39.985,157.464
C08788=1034.090,-69.232,-82.035,168.106,39.986,157.464
C08789=1034.083,-69.482,-82.023,168.103,39.986,157.464
C08790=1034.078,-69.732,-82.012,168.101,39.987,157.464
C08791=1034.071,-69.981,-82.000,168.099,39.988,157.464
C08792=1034.065,-70.232,-81.988,168.096,39.989,157.464
C08793=1034.059,-70.481,-81.976,168.094,39.989,157.464
C08794=1034.053,-70.731,-81.965,168.091,39.990,157.464
C08795=1034.047,-70.980,-81.954,168.088,39.991,157.464
C08796=1034.041,-71.230,-81.942,168.085,39.992,157.464
C08797=1034.036,-71.480,-81.931,168.083,39.992,157.464
C08798=1034.029,-71.729,-81.919,168.080,39.993,157.464
C08799=1034.023,-71.979,-81.908,168.077,39.994,157.464
C08800=1034.017,-72.229,-81.897,168.075,39.995,157.465
C08801=1034.011,-72.478,-81.885,168.072,39.995,157.464
C08802=1034.006,-72.727,-81.874,168.069,39.996,157.464
C08803=1034.000,-72.978,-81.862,168.066,39.997,157.465
C08804=1033.994,-73.227,-81.851,168.065,39.998,157.465
C08805=1033.987,-73.477,-81.840,168.061,39.998,157.465
C08806=1033.981,-73.726,-81.829,168.059,39.999,157.465
C08807=1033.975,-73.976,-81.817,168.057,40.000,157.465
C08808=1033.970,-74.226,-81.805,168.054,40.001,157.465
C08809=1033.963,-74.475,-81.795,168.051,40.002,157.465
C08810=1033.957,-74.725,-81.784,168.048,40.003,157.465
C08811=1033.951,-74.975,-81.773,168.046,40.003,157.465
C08812=1033.945,-75.224,-81.761,168.043,40.004,157.465
C08813=1033.938,-75.474,-81.750,168.040,40.005,157.465
C08814=1033.933,-75.724,-81.739,168.037,40.006,157.465
C08815=1033.926,-75.974,-81.728,168.035,40.007,157.465
C08816=1033.920,-76.223,-81.717,168.033,40.008,157.465
C08817=1033.914,-76.472,-81.705,168.030,40.009,157.465
C08818=1033.908,-76.722,-81.694,168.027,40.009,157.465
C08819=1033.902,-76.972,-81.683,168.024,40.010,157.465
C08820=1033.895,-77.222,-81.672,168.022,40.011,157.465
C08821=1033.890,-77.471,-81.661,168.019,40.012,157.465
C08822=1033.883,-77.722,-81.650,168.016,40.013,157.465
///RCONF 1,0,0,0,1,0,0,0,0,0,0,0,0,0,0,0,0,0,0,0,0,0,0,0
C08823=1033.877,-77.971,-81.639,168.013,40.014,157.465
C08824=1033.872,-78.220,-81.628,168.010,40.015,157.465
C08825=1033.865,-78.471,-81.617,168.008,40.016,157.465
C08826=1033.859,-78.720,-81.606,168.006,40.017,157.466
C08827=1033.853,-78.970,-81.594,168.003,40.017,157.466
C08828=1033.847,-79.219,-81.583,168.000,40.018,157.466
C08829=1033.841,-79.468,-81.573,167.998,40.019,157.466
C08830=1033.834,-79.719,-81.562,167.995,40.020,157.466
C08831=1033.829,-79.968,-81.551,167.992,40.021,157.466
C08832=1033.823,-80.218,-81.540,167.989,40.022,157.466
C08833=1033.817,-80.468,-81.529,167.986,40.023,157.466
C08834=1033.810,-80.717,-81.519,167.984,40.025,157.466
C08835=1033.804,-80.967,-81.507,167.982,40.025,157.466
C08836=1033.797,-81.216,-81.497,167.979,40.026,157.466
C08837=1033.792,-81.466,-81.487,167.976,40.027,157.466
C08838=1033.786,-81.717,-81.476,167.973,40.028,157.466
C08839=1033.779,-81.966,-81.465,167.970,40.029,157.466
C08840=1033.773,-82.215,-81.455,167.968,40.030,157.466
C08841=1033.767,-82.465,-81.443,167.965,40.032,157.467
C08842=1033.760,-82.715,-81.433,167.962,40.033,157.467
C08843=1033.755,-82.964,-81.422,167.960,40.034,157.467
C08844=1033.748,-83.214,-81.411,167.957,40.034,157.467
C08845=1033.742,-83.464,-81.401,167.954,40.035,157.467
C08846=1033.737,-83.714,-81.391,167.952,40.036,157.467
C08847=1033.729,-83.998,-81.377,167.948,40.038,157.467
C08848=1033.722,-84.283,-81.366,167.945,40.039,157.467
C08849=1033.715,-84.568,-81.353,167.942,40.040,157.467
C08850=1033.708,-84.853,-81.341,167.940,40.041,157.467
C08851=1033.702,-85.102,-81.331,167.937,40.042,157.467
C08852=1033.696,-85.353,-81.321,167.934,40.043,157.467
C08853=1033.689,-85.602,-81.310,167.931,40.044,157.467
C08854=1033.683,-85.852,-81.299,167.928,40.045,157.467
C08855=1033.678,-86.101,-81.288,167.925,40.047,157.468
C08856=1033.671,-86.351,-81.278,167.923,40.048,157.468
C08857=1033.665,-86.601,-81.268,167.920,40.049,157.468
C08858=1033.659,-86.851,-81.257,167.917,40.050,157.468
C08859=1033.653,-87.100,-81.247,167.915,40.050,157.468
C08860=1033.647,-87.350,-81.235,167.912,40.052,157.468
C08861=1033.640,-87.600,-81.226,167.909,40.053,157.468
C08862=1033.635,-87.849,-81.215,167.906,40.054,157.468
C08863=1033.628,-88.098,-81.205,167.904,40.055,157.468
C08864=1033.622,-88.349,-81.194,167.901,40.056,157.468
C08865=1033.616,-88.599,-81.183,167.898,40.057,157.468
C08866=1033.610,-88.848,-81.173,167.896,40.058,157.468
C08867=1033.604,-89.098,-81.163,167.893,40.059,157.468
C08868=1033.598,-89.347,-81.152,167.890,40.060,157.468
C08869=1033.592,-89.597,-81.141,167.887,40.061,157.468
C08870=1033.586,-89.848,-81.131,167.885,40.062,157.469
C08871=1033.580,-90.097,-81.121,167.882,40.064,157.469
C08872=1033.574,-90.346,-81.110,167.879,40.065,157.469
C08873=1033.568,-90.596,-81.100,167.876,40.065,157.469
C08874=1033.562,-90.845,-81.089,167.874,40.066,157.469
C08875=1033.556,-91.095,-81.080,167.871,40.067,157.469
C08876=1033.550,-91.345,-81.069,167.869,40.069,157.469
C08877=1033.544,-91.595,-81.058,167.866,40.070,157.469
C08878=1033.538,-91.845,-81.048,167.863,40.071,157.469
C08879=1033.532,-92.094,-81.037,167.860,40.072,157.469
C08880=1033.526,-92.344,-81.028,167.857,40.073,157.469
C08881=1033.520,-92.594,-81.017,167.855,40.074,157.469
C08882=1033.514,-92.843,-81.007,167.852,40.075,157.469
C08883=1033.508,-93.093,-80.996,167.850,40.076,157.470
C08884=1033.501,-93.343,-80.986,167.847,40.077,157.470
C08885=1033.496,-93.593,-80.976,167.844,40.078,157.470
C08886=1033.490,-93.843,-80.965,167.841,40.080,157.470
C08887=1033.484,-94.092,-80.955,167.838,40.081,157.470
C08888=1033.478,-94.342,-80.945,167.835,40.081,157.470
C08889=1033.472,-94.591,-80.935,167.832,40.082,157.470
C08890=1033.466,-94.841,-80.925,167.831,40.083,157.470
C08891=1033.460,-95.091,-80.914,167.828,40.085,157.470
C08892=1033.454,-95.341,-80.904,167.825,40.086,157.470
C08893=1033.448,-95.590,-80.894,167.822,40.087,157.470
C08894=1033.443,-95.840,-80.884,167.819,40.088,157.470
C08895=1033.436,-96.089,-80.873,167.816,40.089,157.470
C08896=1033.431,-96.339,-80.863,167.813,40.090,157.471
C08897=1033.424,-96.589,-80.854,167.811,40.091,157.471
C08898=1033.419,-96.839,-80.843,167.809,40.092,157.471
C08899=1033.413,-97.088,-80.833,167.806,40.093,157.471
C08900=1033.407,-97.338,-80.822,167.803,40.095,157.471
C08901=1033.401,-97.588,-80.813,167.800,40.096,157.471
C08902=1033.395,-97.838,-80.803,167.797,40.097,157.471
C08903=1033.389,-98.087,-80.792,167.794,40.098,157.471
C08904=1033.383,-98.337,-80.783,167.792,40.099,157.471
C08905=1033.377,-98.587,-80.773,167.789,40.101,157.471
C08906=1033.371,-98.837,-80.763,167.786,40.102,157.471
C08907=1033.364,-99.086,-80.753,167.784,40.103,157.471
C08908=1033.358,-99.336,-80.743,167.781,40.104,157.472
C08909=1033.353,-99.586,-80.733,167.778,40.105,157.472
C08910=1033.347,-99.836,-80.723,167.776,40.107,157.472
C08911=1033.339,-100.122,-80.711,167.772,40.108,157.472
C08912=1033.332,-100.410,-80.700,167.769,40.109,157.472
C08913=1033.326,-100.697,-80.689,167.766,40.111,157.472
C08914=1033.318,-100.984,-80.678,167.762,40.112,157.472
C08915=1033.312,-101.234,-80.668,167.759,40.114,157.472
C08916=1033.307,-101.484,-80.658,167.757,40.115,157.472
C08917=1033.301,-101.734,-80.648,167.755,40.115,157.472
C08918=1033.294,-101.983,-80.638,167.752,40.117,157.473
C08919=1033.288,-102.233,-80.628,167.749,40.118,157.473
C08920=1033.283,-102.483,-80.618,167.746,40.120,157.473
C08921=1033.276,-102.732,-80.609,167.743,40.121,157.473
C08922=1033.270,-102.982,-80.599,167.741,40.122,157.473
C08923=1033.265,-103.231,-80.590,167.738,40.123,157.473
C08924=1033.259,-103.481,-80.580,167.735,40.125,157.473
C08925=1033.253,-103.731,-80.569,167.732,40.126,157.473
C08926=1033.247,-103.980,-80.560,167.729,40.127,157.473
C08927=1033.240,-104.230,-80.550,167.726,40.128,157.473
C08928=1033.234,-104.480,-80.541,167.723,40.129,157.474
C08929=1033.229,-104.730,-80.531,167.721,40.131,157.474
C08930=1033.223,-104.980,-80.521,167.719,40.132,157.474
C08931=1033.217,-105.230,-80.511,167.716,40.133,157.474
C08932=1033.211,-105.479,-80.502,167.713,40.134,157.474
C08933=1033.205,-105.729,-80.493,167.710,40.136,157.474
C08934=1033.199,-105.979,-80.482,167.708,40.137,157.474
C08935=1033.193,-106.229,-80.473,167.705,40.138,157.474
C08936=1033.187,-106.478,-80.463,167.702,40.139,157.474
C08937=1033.181,-106.728,-80.454,167.699,40.141,157.475
C08938=1033.175,-106.977,-80.445,167.696,40.142,157.475
C08939=1033.169,-107.227,-80.435,167.693,40.144,157.475
C08940=1033.164,-107.477,-80.425,167.691,40.145,157.475
C08941=1033.157,-107.727,-80.415,167.688,40.146,157.475
C08942=1033.151,-107.977,-80.406,167.685,40.147,157.475
C08943=1033.145,-108.227,-80.396,167.682,40.149,157.475
C08944=1033.140,-108.476,-80.387,167.679,40.150,157.475
C08945=1033.133,-108.725,-80.377,167.676,40.151,157.475
C08946=1033.128,-108.976,-80.369,167.674,40.153,157.476
C08947=1033.121,-109.226,-80.359,167.671,40.154,157.476
C08948=1033.115,-109.475,-80.349,167.668,40.156,157.476
C08949=1033.109,-109.725,-80.340,167.665,40.157,157.476
C08950=1033.103,-109.974,-80.331,167.662,40.158,157.476
C08951=1033.097,-110.224,-80.321,167.660,40.160,157.476
C08952=1033.091,-110.474,-80.312,167.658,40.161,157.476
C08953=1033.085,-110.724,-80.303,167.655,40.162,157.476
C08954=1033.080,-110.973,-80.293,167.652,40.164,157.476
C08955=1033.073,-111.223,-80.284,167.649,40.165,157.477
C08956=1033.067,-111.473,-80.274,167.647,40.166,157.477
C08957=1033.061,-111.723,-80.265,167.644,40.168,157.477
C08958=1033.056,-111.973,-80.256,167.641,40.169,157.477
C08959=1033.050,-112.222,-80.247,167.638,40.171,157.477
C08960=1033.044,-112.472,-80.237,167.635,40.172,157.477
C08961=1033.037,-112.722,-80.228,167.632,40.173,157.477
C08962=1033.032,-112.972,-80.219,167.630,40.175,157.477
C08963=1033.026,-113.221,-80.210,167.627,40.176,157.477
C08964=1033.020,-113.471,-80.200,167.624,40.177,157.478
C08965=1033.014,-113.720,-80.191,167.621,40.179,157.478
C08966=1033.008,-113.971,-80.182,167.618,40.180,157.478
C08967=1033.002,-114.221,-80.172,167.616,40.182,157.478
C08968=1032.997,-114.470,-80.163,167.613,40.183,157.478
C08969=1032.991,-114.720,-80.154,167.610,40.184,157.478
C08970=1032.985,-114.970,-80.145,167.607,40.186,157.478
C08971=1032.978,-115.220,-80.135,167.604,40.187,157.478
C08972=1032.973,-115.469,-80.127,167.602,40.188,157.479
C08973=1032.966,-115.719,-80.118,167.599,40.190,157.479
C08974=1032.960,-115.969,-80.108,167.596,40.192,157.479
C08975=1032.954,-116.255,-80.098,167.593,40.193,157.479
C08976=1032.948,-116.542,-80.087,167.589,40.195,157.479
C08977=1032.940,-116.828,-80.077,167.587,40.197,157.479
C08978=1032.933,-117.115,-80.066,167.583,40.198,157.479
C08979=1032.928,-117.364,-80.058,167.580,40.200,157.480
C08980=1032.922,-117.614,-80.048,167.577,40.201,157.480
C08981=1032.915,-117.864,-80.040,167.574,40.203,157.480
C08982=1032.910,-118.113,-80.031,167.572,40.204,157.480
C08983=1032.904,-118.363,-80.021,167.569,40.206,157.480
C08984=1032.898,-118.614,-80.012,167.566,40.207,157.480
C08985=1032.892,-118.863,-80.003,167.563,40.208,157.480
C08986=1032.886,-119.113,-79.994,167.561,40.210,157.480
C08987=1032.880,-119.362,-79.986,167.558,40.212,157.481
C08988=1032.874,-119.612,-79.977,167.555,40.213,157.481
C08989=1032.868,-119.862,-79.967,167.552,40.214,157.481
C08990=1032.863,-120.112,-79.959,167.549,40.216,157.481
C08991=1032.857,-120.362,-79.950,167.547,40.218,157.481
C08992=1032.850,-120.611,-79.941,167.544,40.219,157.481
C08993=1032.845,-120.861,-79.933,167.541,40.220,157.481
C08994=1032.839,-121.111,-79.923,167.538,40.222,157.482
C08995=1032.833,-121.361,-79.914,167.535,40.223,157.482
C08996=1032.827,-121.610,-79.906,167.533,40.225,157.482
C08997=1032.821,-121.860,-79.897,167.530,40.227,157.482
C08998=1032.815,-122.111,-79.888,167.527,40.228,157.482
C08999=1032.810,-122.360,-79.879,167.524,40.229,157.482
C09000=1032.803,-122.610,-79.871,167.521,40.231,157.482
C09001=1032.797,-122.859,-79.862,167.519,40.233,157.482
C09002=1032.792,-123.109,-79.853,167.516,40.234,157.483
C09003=1032.786,-123.359,-79.844,167.513,40.236,157.483
C09004=1032.780,-123.609,-79.835,167.510,40.237,157.483
C09005=1032.774,-123.858,-79.827,167.508,40.238,157.483
C09006=1032.768,-124.109,-79.818,167.505,40.240,157.483
C09007=1032.763,-124.358,-79.809,167.502,40.242,157.483
C09008=1032.756,-124.608,-79.800,167.499,40.243,157.483
C09009=1032.751,-124.858,-79.792,167.497,40.245,157.484
C09010=1032.745,-125.108,-79.783,167.494,40.247,157.484
C09011=1032.739,-125.357,-79.774,167.491,40.248,157.484
C09012=1032.733,-125.607,-79.766,167.488,40.250,157.484
C09013=1032.727,-125.857,-79.757,167.485,40.252,157.484
C09014=1032.721,-126.107,-79.749,167.483,40.253,157.484
C09015=1032.715,-126.356,-79.740,167.480,40.255,157.485
C09016=1032.709,-126.606,-79.732,167.477,40.256,157.485
C09017=1032.703,-126.856,-79.723,167.474,40.257,157.485
C09018=1032.698,-127.106,-79.714,167.472,40.259,157.485
C09019=1032.691,-127.355,-79.705,167.469,40.261,157.485
C09020=1032.686,-127.605,-79.697,167.466,40.262,157.485
C09021=1032.680,-127.854,-79.689,167.463,40.264,157.485
C09022=1032.675,-128.104,-79.679,167.460,40.266,157.486
C09023=1032.671,-128.354,-79.670,167.457,40.266,157.485
C09024=1032.667,-128.603,-79.660,167.454,40.266,157.485
C09025=1032.662,-128.853,-79.649,167.452,40.266,157.485
C09026=1032.660,-129.103,-79.638,167.450,40.266,157.485
C09027=1032.658,-129.353,-79.625,167.448,40.265,157.485
C09028=1032.657,-129.603,-79.614,167.445,40.263,157.484
C09029=1032.656,-129.852,-79.600,167.444,40.261,157.484
C09030=1032.656,-130.102,-79.587,167.441,40.258,157.484
